;FOLD SLIN P127 Vel=2 m/s CPDAT127 Tool[4]:Microflown3D Base[2]:straight_sol;%{PE}
;FOLD Parameters ;%{h}
;Params IlfProvider=kukaroboter.basistech.inlineforms.movement.spline; Kuka.IsGlobalPoint=False; Kuka.PointName=P127; Kuka.BlendingEnabled=False; Kuka.MoveDataName=CPDAT127; Kuka.VelocityPath=2.000; Kuka.VelocityFieldEnabled=True; Kuka.ColDetectFieldEnabled=True; Kuka.CurrentCDSetIndex=0; Kuka.MovementParameterFieldEnabled=True; IlfCommand=SLIN
;ENDFOLD
SLIN XP127 WITH $VEL = SVEL_CP(2.0, , LCPDAT127),$TOOL = STOOL2(FP127),$BASE = SBASE(FP127.BASE_NO),$IPO_MODE = SIPO_MODE(FP127.IPO_FRAME),$LOAD = SLOAD(FP127.TOOL_NO),$ACC = SACC_CP(LCPDAT127),$ORI_TYPE = SORI_TYP(LCPDAT127),$APO = SAPO(LCPDAT127),$JERK = SJERK(LCPDAT127),$COLLMON_TOL_PRO[1] = USE_CM_PRO_VALUES(0)
;ENDFOLD

;FOLD SLIN P128 Vel=2 m/s CPDAT128 Tool[4]:Microflown3D Base[2]:straight_sol;%{PE}
;FOLD Parameters ;%{h}
;Params IlfProvider=kukaroboter.basistech.inlineforms.movement.spline; Kuka.IsGlobalPoint=False; Kuka.PointName=P128; Kuka.BlendingEnabled=False; Kuka.MoveDataName=CPDAT128; Kuka.VelocityPath=2.000; Kuka.VelocityFieldEnabled=True; Kuka.ColDetectFieldEnabled=True; Kuka.CurrentCDSetIndex=0; Kuka.MovementParameterFieldEnabled=True; IlfCommand=SLIN
;ENDFOLD
SLIN XP128 WITH $VEL = SVEL_CP(2.0, , LCPDAT128),$TOOL = STOOL2(FP128),$BASE = SBASE(FP128.BASE_NO),$IPO_MODE = SIPO_MODE(FP128.IPO_FRAME),$LOAD = SLOAD(FP128.TOOL_NO),$ACC = SACC_CP(LCPDAT128),$ORI_TYPE = SORI_TYP(LCPDAT128),$APO = SAPO(LCPDAT128),$JERK = SJERK(LCPDAT128),$COLLMON_TOL_PRO[1] = USE_CM_PRO_VALUES(0)
;ENDFOLD

;FOLD SLIN P129 Vel=2 m/s CPDAT129 Tool[4]:Microflown3D Base[2]:straight_sol;%{PE}
;FOLD Parameters ;%{h}
;Params IlfProvider=kukaroboter.basistech.inlineforms.movement.spline; Kuka.IsGlobalPoint=False; Kuka.PointName=P129; Kuka.BlendingEnabled=False; Kuka.MoveDataName=CPDAT129; Kuka.VelocityPath=2.000; Kuka.VelocityFieldEnabled=True; Kuka.ColDetectFieldEnabled=True; Kuka.CurrentCDSetIndex=0; Kuka.MovementParameterFieldEnabled=True; IlfCommand=SLIN
;ENDFOLD
SLIN XP129 WITH $VEL = SVEL_CP(2.0, , LCPDAT129),$TOOL = STOOL2(FP129),$BASE = SBASE(FP129.BASE_NO),$IPO_MODE = SIPO_MODE(FP129.IPO_FRAME),$LOAD = SLOAD(FP129.TOOL_NO),$ACC = SACC_CP(LCPDAT129),$ORI_TYPE = SORI_TYP(LCPDAT129),$APO = SAPO(LCPDAT129),$JERK = SJERK(LCPDAT129),$COLLMON_TOL_PRO[1] = USE_CM_PRO_VALUES(0)
;ENDFOLD

;FOLD SLIN P130 Vel=2 m/s CPDAT130 Tool[4]:Microflown3D Base[2]:straight_sol;%{PE}
;FOLD Parameters ;%{h}
;Params IlfProvider=kukaroboter.basistech.inlineforms.movement.spline; Kuka.IsGlobalPoint=False; Kuka.PointName=P130; Kuka.BlendingEnabled=False; Kuka.MoveDataName=CPDAT130; Kuka.VelocityPath=2.000; Kuka.VelocityFieldEnabled=True; Kuka.ColDetectFieldEnabled=True; Kuka.CurrentCDSetIndex=0; Kuka.MovementParameterFieldEnabled=True; IlfCommand=SLIN
;ENDFOLD
SLIN XP130 WITH $VEL = SVEL_CP(2.0, , LCPDAT130),$TOOL = STOOL2(FP130),$BASE = SBASE(FP130.BASE_NO),$IPO_MODE = SIPO_MODE(FP130.IPO_FRAME),$LOAD = SLOAD(FP130.TOOL_NO),$ACC = SACC_CP(LCPDAT130),$ORI_TYPE = SORI_TYP(LCPDAT130),$APO = SAPO(LCPDAT130),$JERK = SJERK(LCPDAT130),$COLLMON_TOL_PRO[1] = USE_CM_PRO_VALUES(0)
;ENDFOLD

;FOLD SLIN P131 Vel=2 m/s CPDAT131 Tool[4]:Microflown3D Base[2]:straight_sol;%{PE}
;FOLD Parameters ;%{h}
;Params IlfProvider=kukaroboter.basistech.inlineforms.movement.spline; Kuka.IsGlobalPoint=False; Kuka.PointName=P131; Kuka.BlendingEnabled=False; Kuka.MoveDataName=CPDAT131; Kuka.VelocityPath=2.000; Kuka.VelocityFieldEnabled=True; Kuka.ColDetectFieldEnabled=True; Kuka.CurrentCDSetIndex=0; Kuka.MovementParameterFieldEnabled=True; IlfCommand=SLIN
;ENDFOLD
SLIN XP131 WITH $VEL = SVEL_CP(2.0, , LCPDAT131),$TOOL = STOOL2(FP131),$BASE = SBASE(FP131.BASE_NO),$IPO_MODE = SIPO_MODE(FP131.IPO_FRAME),$LOAD = SLOAD(FP131.TOOL_NO),$ACC = SACC_CP(LCPDAT131),$ORI_TYPE = SORI_TYP(LCPDAT131),$APO = SAPO(LCPDAT131),$JERK = SJERK(LCPDAT131),$COLLMON_TOL_PRO[1] = USE_CM_PRO_VALUES(0)
;ENDFOLD

;FOLD SLIN P132 Vel=2 m/s CPDAT132 Tool[4]:Microflown3D Base[2]:straight_sol;%{PE}
;FOLD Parameters ;%{h}
;Params IlfProvider=kukaroboter.basistech.inlineforms.movement.spline; Kuka.IsGlobalPoint=False; Kuka.PointName=P132; Kuka.BlendingEnabled=False; Kuka.MoveDataName=CPDAT132; Kuka.VelocityPath=2.000; Kuka.VelocityFieldEnabled=True; Kuka.ColDetectFieldEnabled=True; Kuka.CurrentCDSetIndex=0; Kuka.MovementParameterFieldEnabled=True; IlfCommand=SLIN
;ENDFOLD
SLIN XP132 WITH $VEL = SVEL_CP(2.0, , LCPDAT132),$TOOL = STOOL2(FP132),$BASE = SBASE(FP132.BASE_NO),$IPO_MODE = SIPO_MODE(FP132.IPO_FRAME),$LOAD = SLOAD(FP132.TOOL_NO),$ACC = SACC_CP(LCPDAT132),$ORI_TYPE = SORI_TYP(LCPDAT132),$APO = SAPO(LCPDAT132),$JERK = SJERK(LCPDAT132),$COLLMON_TOL_PRO[1] = USE_CM_PRO_VALUES(0)
;ENDFOLD

;FOLD SLIN P133 Vel=2 m/s CPDAT133 Tool[4]:Microflown3D Base[2]:straight_sol;%{PE}
;FOLD Parameters ;%{h}
;Params IlfProvider=kukaroboter.basistech.inlineforms.movement.spline; Kuka.IsGlobalPoint=False; Kuka.PointName=P133; Kuka.BlendingEnabled=False; Kuka.MoveDataName=CPDAT133; Kuka.VelocityPath=2.000; Kuka.VelocityFieldEnabled=True; Kuka.ColDetectFieldEnabled=True; Kuka.CurrentCDSetIndex=0; Kuka.MovementParameterFieldEnabled=True; IlfCommand=SLIN
;ENDFOLD
SLIN XP133 WITH $VEL = SVEL_CP(2.0, , LCPDAT133),$TOOL = STOOL2(FP133),$BASE = SBASE(FP133.BASE_NO),$IPO_MODE = SIPO_MODE(FP133.IPO_FRAME),$LOAD = SLOAD(FP133.TOOL_NO),$ACC = SACC_CP(LCPDAT133),$ORI_TYPE = SORI_TYP(LCPDAT133),$APO = SAPO(LCPDAT133),$JERK = SJERK(LCPDAT133),$COLLMON_TOL_PRO[1] = USE_CM_PRO_VALUES(0)
;ENDFOLD

;FOLD SLIN P134 Vel=2 m/s CPDAT134 Tool[4]:Microflown3D Base[2]:straight_sol;%{PE}
;FOLD Parameters ;%{h}
;Params IlfProvider=kukaroboter.basistech.inlineforms.movement.spline; Kuka.IsGlobalPoint=False; Kuka.PointName=P134; Kuka.BlendingEnabled=False; Kuka.MoveDataName=CPDAT134; Kuka.VelocityPath=2.000; Kuka.VelocityFieldEnabled=True; Kuka.ColDetectFieldEnabled=True; Kuka.CurrentCDSetIndex=0; Kuka.MovementParameterFieldEnabled=True; IlfCommand=SLIN
;ENDFOLD
SLIN XP134 WITH $VEL = SVEL_CP(2.0, , LCPDAT134),$TOOL = STOOL2(FP134),$BASE = SBASE(FP134.BASE_NO),$IPO_MODE = SIPO_MODE(FP134.IPO_FRAME),$LOAD = SLOAD(FP134.TOOL_NO),$ACC = SACC_CP(LCPDAT134),$ORI_TYPE = SORI_TYP(LCPDAT134),$APO = SAPO(LCPDAT134),$JERK = SJERK(LCPDAT134),$COLLMON_TOL_PRO[1] = USE_CM_PRO_VALUES(0)
;ENDFOLD

;FOLD SLIN P135 Vel=1 m/s CPDAT135 Tool[4]:Microflown3D Base[2]:straight_sol;%{PE}
;FOLD Parameters ;%{h}
;Params IlfProvider=kukaroboter.basistech.inlineforms.movement.spline; Kuka.IsGlobalPoint=False; Kuka.PointName=P135; Kuka.BlendingEnabled=False; Kuka.MoveDataName=CPDAT135; Kuka.VelocityPath=1.000; Kuka.VelocityFieldEnabled=True; Kuka.ColDetectFieldEnabled=True; Kuka.CurrentCDSetIndex=0; Kuka.MovementParameterFieldEnabled=True; IlfCommand=SLIN
;ENDFOLD
SLIN XP135 WITH $VEL = SVEL_CP(2.0, , LCPDAT135),$TOOL = STOOL2(FP135),$BASE = SBASE(FP135.BASE_NO),$IPO_MODE = SIPO_MODE(FP135.IPO_FRAME),$LOAD = SLOAD(FP135.TOOL_NO),$ACC = SACC_CP(LCPDAT135),$ORI_TYPE = SORI_TYP(LCPDAT135),$APO = SAPO(LCPDAT135),$JERK = SJERK(LCPDAT135),$COLLMON_TOL_PRO[1] = USE_CM_PRO_VALUES(0)
;ENDFOLD

;FOLD SLIN P136 Vel=1 m/s CPDAT136 Tool[4]:Microflown3D Base[2]:straight_sol;%{PE}
;FOLD Parameters ;%{h}
;Params IlfProvider=kukaroboter.basistech.inlineforms.movement.spline; Kuka.IsGlobalPoint=False; Kuka.PointName=P136; Kuka.BlendingEnabled=False; Kuka.MoveDataName=CPDAT136; Kuka.VelocityPath=1.000; Kuka.VelocityFieldEnabled=True; Kuka.ColDetectFieldEnabled=True; Kuka.CurrentCDSetIndex=0; Kuka.MovementParameterFieldEnabled=True; IlfCommand=SLIN
;ENDFOLD
SLIN XP136 WITH $VEL = SVEL_CP(2.0, , LCPDAT136),$TOOL = STOOL2(FP136),$BASE = SBASE(FP136.BASE_NO),$IPO_MODE = SIPO_MODE(FP136.IPO_FRAME),$LOAD = SLOAD(FP136.TOOL_NO),$ACC = SACC_CP(LCPDAT136),$ORI_TYPE = SORI_TYP(LCPDAT136),$APO = SAPO(LCPDAT136),$JERK = SJERK(LCPDAT136),$COLLMON_TOL_PRO[1] = USE_CM_PRO_VALUES(0)
;ENDFOLD

;FOLD SLIN P137 Vel=2 m/s CPDAT137 Tool[4]:Microflown3D Base[2]:straight_sol;%{PE}
;FOLD Parameters ;%{h}
;Params IlfProvider=kukaroboter.basistech.inlineforms.movement.spline; Kuka.IsGlobalPoint=False; Kuka.PointName=P137; Kuka.BlendingEnabled=False; Kuka.MoveDataName=CPDAT137; Kuka.VelocityPath=2.000; Kuka.VelocityFieldEnabled=True; Kuka.ColDetectFieldEnabled=True; Kuka.CurrentCDSetIndex=0; Kuka.MovementParameterFieldEnabled=True; IlfCommand=SLIN
;ENDFOLD
SLIN XP137 WITH $VEL = SVEL_CP(2.0, , LCPDAT137),$TOOL = STOOL2(FP137),$BASE = SBASE(FP137.BASE_NO),$IPO_MODE = SIPO_MODE(FP137.IPO_FRAME),$LOAD = SLOAD(FP137.TOOL_NO),$ACC = SACC_CP(LCPDAT137),$ORI_TYPE = SORI_TYP(LCPDAT137),$APO = SAPO(LCPDAT137),$JERK = SJERK(LCPDAT137),$COLLMON_TOL_PRO[1] = USE_CM_PRO_VALUES(0)
;ENDFOLD

;FOLD SLIN P138 Vel=2 m/s CPDAT138 Tool[4]:Microflown3D Base[2]:straight_sol;%{PE}
;FOLD Parameters ;%{h}
;Params IlfProvider=kukaroboter.basistech.inlineforms.movement.spline; Kuka.IsGlobalPoint=False; Kuka.PointName=P138; Kuka.BlendingEnabled=False; Kuka.MoveDataName=CPDAT138; Kuka.VelocityPath=2.000; Kuka.VelocityFieldEnabled=True; Kuka.ColDetectFieldEnabled=True; Kuka.CurrentCDSetIndex=0; Kuka.MovementParameterFieldEnabled=True; IlfCommand=SLIN
;ENDFOLD
SLIN XP138 WITH $VEL = SVEL_CP(2.0, , LCPDAT138),$TOOL = STOOL2(FP138),$BASE = SBASE(FP138.BASE_NO),$IPO_MODE = SIPO_MODE(FP138.IPO_FRAME),$LOAD = SLOAD(FP138.TOOL_NO),$ACC = SACC_CP(LCPDAT138),$ORI_TYPE = SORI_TYP(LCPDAT138),$APO = SAPO(LCPDAT138),$JERK = SJERK(LCPDAT138),$COLLMON_TOL_PRO[1] = USE_CM_PRO_VALUES(0)
;ENDFOLD

;FOLD SLIN P139 Vel=2 m/s CPDAT139 Tool[4]:Microflown3D Base[2]:straight_sol;%{PE}
;FOLD Parameters ;%{h}
;Params IlfProvider=kukaroboter.basistech.inlineforms.movement.spline; Kuka.IsGlobalPoint=False; Kuka.PointName=P139; Kuka.BlendingEnabled=False; Kuka.MoveDataName=CPDAT139; Kuka.VelocityPath=2.000; Kuka.VelocityFieldEnabled=True; Kuka.ColDetectFieldEnabled=True; Kuka.CurrentCDSetIndex=0; Kuka.MovementParameterFieldEnabled=True; IlfCommand=SLIN
;ENDFOLD
SLIN XP139 WITH $VEL = SVEL_CP(2.0, , LCPDAT139),$TOOL = STOOL2(FP139),$BASE = SBASE(FP139.BASE_NO),$IPO_MODE = SIPO_MODE(FP139.IPO_FRAME),$LOAD = SLOAD(FP139.TOOL_NO),$ACC = SACC_CP(LCPDAT139),$ORI_TYPE = SORI_TYP(LCPDAT139),$APO = SAPO(LCPDAT139),$JERK = SJERK(LCPDAT139),$COLLMON_TOL_PRO[1] = USE_CM_PRO_VALUES(0)
;ENDFOLD

;FOLD SLIN P140 Vel=2 m/s CPDAT140 Tool[4]:Microflown3D Base[2]:straight_sol;%{PE}
;FOLD Parameters ;%{h}
;Params IlfProvider=kukaroboter.basistech.inlineforms.movement.spline; Kuka.IsGlobalPoint=False; Kuka.PointName=P140; Kuka.BlendingEnabled=False; Kuka.MoveDataName=CPDAT140; Kuka.VelocityPath=2.000; Kuka.VelocityFieldEnabled=True; Kuka.ColDetectFieldEnabled=True; Kuka.CurrentCDSetIndex=0; Kuka.MovementParameterFieldEnabled=True; IlfCommand=SLIN
;ENDFOLD
SLIN XP140 WITH $VEL = SVEL_CP(2.0, , LCPDAT140),$TOOL = STOOL2(FP140),$BASE = SBASE(FP140.BASE_NO),$IPO_MODE = SIPO_MODE(FP140.IPO_FRAME),$LOAD = SLOAD(FP140.TOOL_NO),$ACC = SACC_CP(LCPDAT140),$ORI_TYPE = SORI_TYP(LCPDAT140),$APO = SAPO(LCPDAT140),$JERK = SJERK(LCPDAT140),$COLLMON_TOL_PRO[1] = USE_CM_PRO_VALUES(0)
;ENDFOLD

;FOLD SLIN P141 Vel=2 m/s CPDAT141 Tool[4]:Microflown3D Base[2]:straight_sol;%{PE}
;FOLD Parameters ;%{h}
;Params IlfProvider=kukaroboter.basistech.inlineforms.movement.spline; Kuka.IsGlobalPoint=False; Kuka.PointName=P141; Kuka.BlendingEnabled=False; Kuka.MoveDataName=CPDAT141; Kuka.VelocityPath=2.000; Kuka.VelocityFieldEnabled=True; Kuka.ColDetectFieldEnabled=True; Kuka.CurrentCDSetIndex=0; Kuka.MovementParameterFieldEnabled=True; IlfCommand=SLIN
;ENDFOLD
SLIN XP141 WITH $VEL = SVEL_CP(2.0, , LCPDAT141),$TOOL = STOOL2(FP141),$BASE = SBASE(FP141.BASE_NO),$IPO_MODE = SIPO_MODE(FP141.IPO_FRAME),$LOAD = SLOAD(FP141.TOOL_NO),$ACC = SACC_CP(LCPDAT141),$ORI_TYPE = SORI_TYP(LCPDAT141),$APO = SAPO(LCPDAT141),$JERK = SJERK(LCPDAT141),$COLLMON_TOL_PRO[1] = USE_CM_PRO_VALUES(0)
;ENDFOLD

;FOLD SLIN P142 Vel=2 m/s CPDAT142 Tool[4]:Microflown3D Base[2]:straight_sol;%{PE}
;FOLD Parameters ;%{h}
;Params IlfProvider=kukaroboter.basistech.inlineforms.movement.spline; Kuka.IsGlobalPoint=False; Kuka.PointName=P142; Kuka.BlendingEnabled=False; Kuka.MoveDataName=CPDAT142; Kuka.VelocityPath=2.000; Kuka.VelocityFieldEnabled=True; Kuka.ColDetectFieldEnabled=True; Kuka.CurrentCDSetIndex=0; Kuka.MovementParameterFieldEnabled=True; IlfCommand=SLIN
;ENDFOLD
SLIN XP142 WITH $VEL = SVEL_CP(2.0, , LCPDAT142),$TOOL = STOOL2(FP142),$BASE = SBASE(FP142.BASE_NO),$IPO_MODE = SIPO_MODE(FP142.IPO_FRAME),$LOAD = SLOAD(FP142.TOOL_NO),$ACC = SACC_CP(LCPDAT142),$ORI_TYPE = SORI_TYP(LCPDAT142),$APO = SAPO(LCPDAT142),$JERK = SJERK(LCPDAT142),$COLLMON_TOL_PRO[1] = USE_CM_PRO_VALUES(0)
;ENDFOLD

;FOLD SLIN P143 Vel=2 m/s CPDAT143 Tool[4]:Microflown3D Base[2]:straight_sol;%{PE}
;FOLD Parameters ;%{h}
;Params IlfProvider=kukaroboter.basistech.inlineforms.movement.spline; Kuka.IsGlobalPoint=False; Kuka.PointName=P143; Kuka.BlendingEnabled=False; Kuka.MoveDataName=CPDAT143; Kuka.VelocityPath=2.000; Kuka.VelocityFieldEnabled=True; Kuka.ColDetectFieldEnabled=True; Kuka.CurrentCDSetIndex=0; Kuka.MovementParameterFieldEnabled=True; IlfCommand=SLIN
;ENDFOLD
SLIN XP143 WITH $VEL = SVEL_CP(2.0, , LCPDAT143),$TOOL = STOOL2(FP143),$BASE = SBASE(FP143.BASE_NO),$IPO_MODE = SIPO_MODE(FP143.IPO_FRAME),$LOAD = SLOAD(FP143.TOOL_NO),$ACC = SACC_CP(LCPDAT143),$ORI_TYPE = SORI_TYP(LCPDAT143),$APO = SAPO(LCPDAT143),$JERK = SJERK(LCPDAT143),$COLLMON_TOL_PRO[1] = USE_CM_PRO_VALUES(0)
;ENDFOLD

;FOLD SLIN P144 Vel=2 m/s CPDAT144 Tool[4]:Microflown3D Base[2]:straight_sol;%{PE}
;FOLD Parameters ;%{h}
;Params IlfProvider=kukaroboter.basistech.inlineforms.movement.spline; Kuka.IsGlobalPoint=False; Kuka.PointName=P144; Kuka.BlendingEnabled=False; Kuka.MoveDataName=CPDAT144; Kuka.VelocityPath=2.000; Kuka.VelocityFieldEnabled=True; Kuka.ColDetectFieldEnabled=True; Kuka.CurrentCDSetIndex=0; Kuka.MovementParameterFieldEnabled=True; IlfCommand=SLIN
;ENDFOLD
SLIN XP144 WITH $VEL = SVEL_CP(2.0, , LCPDAT144),$TOOL = STOOL2(FP144),$BASE = SBASE(FP144.BASE_NO),$IPO_MODE = SIPO_MODE(FP144.IPO_FRAME),$LOAD = SLOAD(FP144.TOOL_NO),$ACC = SACC_CP(LCPDAT144),$ORI_TYPE = SORI_TYP(LCPDAT144),$APO = SAPO(LCPDAT144),$JERK = SJERK(LCPDAT144),$COLLMON_TOL_PRO[1] = USE_CM_PRO_VALUES(0)
;ENDFOLD

;FOLD SLIN P145 Vel=2 m/s CPDAT145 Tool[4]:Microflown3D Base[2]:straight_sol;%{PE}
;FOLD Parameters ;%{h}
;Params IlfProvider=kukaroboter.basistech.inlineforms.movement.spline; Kuka.IsGlobalPoint=False; Kuka.PointName=P145; Kuka.BlendingEnabled=False; Kuka.MoveDataName=CPDAT145; Kuka.VelocityPath=2.000; Kuka.VelocityFieldEnabled=True; Kuka.ColDetectFieldEnabled=True; Kuka.CurrentCDSetIndex=0; Kuka.MovementParameterFieldEnabled=True; IlfCommand=SLIN
;ENDFOLD
SLIN XP145 WITH $VEL = SVEL_CP(2.0, , LCPDAT145),$TOOL = STOOL2(FP145),$BASE = SBASE(FP145.BASE_NO),$IPO_MODE = SIPO_MODE(FP145.IPO_FRAME),$LOAD = SLOAD(FP145.TOOL_NO),$ACC = SACC_CP(LCPDAT145),$ORI_TYPE = SORI_TYP(LCPDAT145),$APO = SAPO(LCPDAT145),$JERK = SJERK(LCPDAT145),$COLLMON_TOL_PRO[1] = USE_CM_PRO_VALUES(0)
;ENDFOLD

;FOLD SLIN P146 Vel=2 m/s CPDAT146 Tool[4]:Microflown3D Base[2]:straight_sol;%{PE}
;FOLD Parameters ;%{h}
;Params IlfProvider=kukaroboter.basistech.inlineforms.movement.spline; Kuka.IsGlobalPoint=False; Kuka.PointName=P146; Kuka.BlendingEnabled=False; Kuka.MoveDataName=CPDAT146; Kuka.VelocityPath=2.000; Kuka.VelocityFieldEnabled=True; Kuka.ColDetectFieldEnabled=True; Kuka.CurrentCDSetIndex=0; Kuka.MovementParameterFieldEnabled=True; IlfCommand=SLIN
;ENDFOLD
SLIN XP146 WITH $VEL = SVEL_CP(2.0, , LCPDAT146),$TOOL = STOOL2(FP146),$BASE = SBASE(FP146.BASE_NO),$IPO_MODE = SIPO_MODE(FP146.IPO_FRAME),$LOAD = SLOAD(FP146.TOOL_NO),$ACC = SACC_CP(LCPDAT146),$ORI_TYPE = SORI_TYP(LCPDAT146),$APO = SAPO(LCPDAT146),$JERK = SJERK(LCPDAT146),$COLLMON_TOL_PRO[1] = USE_CM_PRO_VALUES(0)
;ENDFOLD

;FOLD SLIN P147 Vel=2 m/s CPDAT147 Tool[4]:Microflown3D Base[2]:straight_sol;%{PE}
;FOLD Parameters ;%{h}
;Params IlfProvider=kukaroboter.basistech.inlineforms.movement.spline; Kuka.IsGlobalPoint=False; Kuka.PointName=P147; Kuka.BlendingEnabled=False; Kuka.MoveDataName=CPDAT147; Kuka.VelocityPath=2.000; Kuka.VelocityFieldEnabled=True; Kuka.ColDetectFieldEnabled=True; Kuka.CurrentCDSetIndex=0; Kuka.MovementParameterFieldEnabled=True; IlfCommand=SLIN
;ENDFOLD
SLIN XP147 WITH $VEL = SVEL_CP(2.0, , LCPDAT147),$TOOL = STOOL2(FP147),$BASE = SBASE(FP147.BASE_NO),$IPO_MODE = SIPO_MODE(FP147.IPO_FRAME),$LOAD = SLOAD(FP147.TOOL_NO),$ACC = SACC_CP(LCPDAT147),$ORI_TYPE = SORI_TYP(LCPDAT147),$APO = SAPO(LCPDAT147),$JERK = SJERK(LCPDAT147),$COLLMON_TOL_PRO[1] = USE_CM_PRO_VALUES(0)
;ENDFOLD

;FOLD SLIN P148 Vel=2 m/s CPDAT148 Tool[4]:Microflown3D Base[2]:straight_sol;%{PE}
;FOLD Parameters ;%{h}
;Params IlfProvider=kukaroboter.basistech.inlineforms.movement.spline; Kuka.IsGlobalPoint=False; Kuka.PointName=P148; Kuka.BlendingEnabled=False; Kuka.MoveDataName=CPDAT148; Kuka.VelocityPath=2.000; Kuka.VelocityFieldEnabled=True; Kuka.ColDetectFieldEnabled=True; Kuka.CurrentCDSetIndex=0; Kuka.MovementParameterFieldEnabled=True; IlfCommand=SLIN
;ENDFOLD
SLIN XP148 WITH $VEL = SVEL_CP(2.0, , LCPDAT148),$TOOL = STOOL2(FP148),$BASE = SBASE(FP148.BASE_NO),$IPO_MODE = SIPO_MODE(FP148.IPO_FRAME),$LOAD = SLOAD(FP148.TOOL_NO),$ACC = SACC_CP(LCPDAT148),$ORI_TYPE = SORI_TYP(LCPDAT148),$APO = SAPO(LCPDAT148),$JERK = SJERK(LCPDAT148),$COLLMON_TOL_PRO[1] = USE_CM_PRO_VALUES(0)
;ENDFOLD

;FOLD SLIN P149 Vel=2 m/s CPDAT149 Tool[4]:Microflown3D Base[2]:straight_sol;%{PE}
;FOLD Parameters ;%{h}
;Params IlfProvider=kukaroboter.basistech.inlineforms.movement.spline; Kuka.IsGlobalPoint=False; Kuka.PointName=P149; Kuka.BlendingEnabled=False; Kuka.MoveDataName=CPDAT149; Kuka.VelocityPath=2.000; Kuka.VelocityFieldEnabled=True; Kuka.ColDetectFieldEnabled=True; Kuka.CurrentCDSetIndex=0; Kuka.MovementParameterFieldEnabled=True; IlfCommand=SLIN
;ENDFOLD
SLIN XP149 WITH $VEL = SVEL_CP(2.0, , LCPDAT149),$TOOL = STOOL2(FP149),$BASE = SBASE(FP149.BASE_NO),$IPO_MODE = SIPO_MODE(FP149.IPO_FRAME),$LOAD = SLOAD(FP149.TOOL_NO),$ACC = SACC_CP(LCPDAT149),$ORI_TYPE = SORI_TYP(LCPDAT149),$APO = SAPO(LCPDAT149),$JERK = SJERK(LCPDAT149),$COLLMON_TOL_PRO[1] = USE_CM_PRO_VALUES(0)
;ENDFOLD

;FOLD SLIN P150 Vel=2 m/s CPDAT150 Tool[4]:Microflown3D Base[2]:straight_sol;%{PE}
;FOLD Parameters ;%{h}
;Params IlfProvider=kukaroboter.basistech.inlineforms.movement.spline; Kuka.IsGlobalPoint=False; Kuka.PointName=P150; Kuka.BlendingEnabled=False; Kuka.MoveDataName=CPDAT150; Kuka.VelocityPath=2.000; Kuka.VelocityFieldEnabled=True; Kuka.ColDetectFieldEnabled=True; Kuka.CurrentCDSetIndex=0; Kuka.MovementParameterFieldEnabled=True; IlfCommand=SLIN
;ENDFOLD
SLIN XP150 WITH $VEL = SVEL_CP(2.0, , LCPDAT150),$TOOL = STOOL2(FP150),$BASE = SBASE(FP150.BASE_NO),$IPO_MODE = SIPO_MODE(FP150.IPO_FRAME),$LOAD = SLOAD(FP150.TOOL_NO),$ACC = SACC_CP(LCPDAT150),$ORI_TYPE = SORI_TYP(LCPDAT150),$APO = SAPO(LCPDAT150),$JERK = SJERK(LCPDAT150),$COLLMON_TOL_PRO[1] = USE_CM_PRO_VALUES(0)
;ENDFOLD

;FOLD SLIN P151 Vel=2 m/s CPDAT151 Tool[4]:Microflown3D Base[2]:straight_sol;%{PE}
;FOLD Parameters ;%{h}
;Params IlfProvider=kukaroboter.basistech.inlineforms.movement.spline; Kuka.IsGlobalPoint=False; Kuka.PointName=P151; Kuka.BlendingEnabled=False; Kuka.MoveDataName=CPDAT151; Kuka.VelocityPath=2.000; Kuka.VelocityFieldEnabled=True; Kuka.ColDetectFieldEnabled=True; Kuka.CurrentCDSetIndex=0; Kuka.MovementParameterFieldEnabled=True; IlfCommand=SLIN
;ENDFOLD
SLIN XP151 WITH $VEL = SVEL_CP(2.0, , LCPDAT151),$TOOL = STOOL2(FP151),$BASE = SBASE(FP151.BASE_NO),$IPO_MODE = SIPO_MODE(FP151.IPO_FRAME),$LOAD = SLOAD(FP151.TOOL_NO),$ACC = SACC_CP(LCPDAT151),$ORI_TYPE = SORI_TYP(LCPDAT151),$APO = SAPO(LCPDAT151),$JERK = SJERK(LCPDAT151),$COLLMON_TOL_PRO[1] = USE_CM_PRO_VALUES(0)
;ENDFOLD

;FOLD SLIN P152 Vel=2 m/s CPDAT152 Tool[4]:Microflown3D Base[2]:straight_sol;%{PE}
;FOLD Parameters ;%{h}
;Params IlfProvider=kukaroboter.basistech.inlineforms.movement.spline; Kuka.IsGlobalPoint=False; Kuka.PointName=P152; Kuka.BlendingEnabled=False; Kuka.MoveDataName=CPDAT152; Kuka.VelocityPath=2.000; Kuka.VelocityFieldEnabled=True; Kuka.ColDetectFieldEnabled=True; Kuka.CurrentCDSetIndex=0; Kuka.MovementParameterFieldEnabled=True; IlfCommand=SLIN
;ENDFOLD
SLIN XP152 WITH $VEL = SVEL_CP(2.0, , LCPDAT152),$TOOL = STOOL2(FP152),$BASE = SBASE(FP152.BASE_NO),$IPO_MODE = SIPO_MODE(FP152.IPO_FRAME),$LOAD = SLOAD(FP152.TOOL_NO),$ACC = SACC_CP(LCPDAT152),$ORI_TYPE = SORI_TYP(LCPDAT152),$APO = SAPO(LCPDAT152),$JERK = SJERK(LCPDAT152),$COLLMON_TOL_PRO[1] = USE_CM_PRO_VALUES(0)
;ENDFOLD

;FOLD SLIN P153 Vel=2 m/s CPDAT153 Tool[4]:Microflown3D Base[2]:straight_sol;%{PE}
;FOLD Parameters ;%{h}
;Params IlfProvider=kukaroboter.basistech.inlineforms.movement.spline; Kuka.IsGlobalPoint=False; Kuka.PointName=P153; Kuka.BlendingEnabled=False; Kuka.MoveDataName=CPDAT153; Kuka.VelocityPath=2.000; Kuka.VelocityFieldEnabled=True; Kuka.ColDetectFieldEnabled=True; Kuka.CurrentCDSetIndex=0; Kuka.MovementParameterFieldEnabled=True; IlfCommand=SLIN
;ENDFOLD
SLIN XP153 WITH $VEL = SVEL_CP(2.0, , LCPDAT153),$TOOL = STOOL2(FP153),$BASE = SBASE(FP153.BASE_NO),$IPO_MODE = SIPO_MODE(FP153.IPO_FRAME),$LOAD = SLOAD(FP153.TOOL_NO),$ACC = SACC_CP(LCPDAT153),$ORI_TYPE = SORI_TYP(LCPDAT153),$APO = SAPO(LCPDAT153),$JERK = SJERK(LCPDAT153),$COLLMON_TOL_PRO[1] = USE_CM_PRO_VALUES(0)
;ENDFOLD

;FOLD SLIN P154 Vel=2 m/s CPDAT154 Tool[4]:Microflown3D Base[2]:straight_sol;%{PE}
;FOLD Parameters ;%{h}
;Params IlfProvider=kukaroboter.basistech.inlineforms.movement.spline; Kuka.IsGlobalPoint=False; Kuka.PointName=P154; Kuka.BlendingEnabled=False; Kuka.MoveDataName=CPDAT154; Kuka.VelocityPath=2.000; Kuka.VelocityFieldEnabled=True; Kuka.ColDetectFieldEnabled=True; Kuka.CurrentCDSetIndex=0; Kuka.MovementParameterFieldEnabled=True; IlfCommand=SLIN
;ENDFOLD
SLIN XP154 WITH $VEL = SVEL_CP(2.0, , LCPDAT154),$TOOL = STOOL2(FP154),$BASE = SBASE(FP154.BASE_NO),$IPO_MODE = SIPO_MODE(FP154.IPO_FRAME),$LOAD = SLOAD(FP154.TOOL_NO),$ACC = SACC_CP(LCPDAT154),$ORI_TYPE = SORI_TYP(LCPDAT154),$APO = SAPO(LCPDAT154),$JERK = SJERK(LCPDAT154),$COLLMON_TOL_PRO[1] = USE_CM_PRO_VALUES(0)
;ENDFOLD

;FOLD SLIN P155 Vel=2 m/s CPDAT155 Tool[4]:Microflown3D Base[2]:straight_sol;%{PE}
;FOLD Parameters ;%{h}
;Params IlfProvider=kukaroboter.basistech.inlineforms.movement.spline; Kuka.IsGlobalPoint=False; Kuka.PointName=P155; Kuka.BlendingEnabled=False; Kuka.MoveDataName=CPDAT155; Kuka.VelocityPath=2.000; Kuka.VelocityFieldEnabled=True; Kuka.ColDetectFieldEnabled=True; Kuka.CurrentCDSetIndex=0; Kuka.MovementParameterFieldEnabled=True; IlfCommand=SLIN
;ENDFOLD
SLIN XP155 WITH $VEL = SVEL_CP(2.0, , LCPDAT155),$TOOL = STOOL2(FP155),$BASE = SBASE(FP155.BASE_NO),$IPO_MODE = SIPO_MODE(FP155.IPO_FRAME),$LOAD = SLOAD(FP155.TOOL_NO),$ACC = SACC_CP(LCPDAT155),$ORI_TYPE = SORI_TYP(LCPDAT155),$APO = SAPO(LCPDAT155),$JERK = SJERK(LCPDAT155),$COLLMON_TOL_PRO[1] = USE_CM_PRO_VALUES(0)
;ENDFOLD

;FOLD SLIN P156 Vel=2 m/s CPDAT156 Tool[4]:Microflown3D Base[2]:straight_sol;%{PE}
;FOLD Parameters ;%{h}
;Params IlfProvider=kukaroboter.basistech.inlineforms.movement.spline; Kuka.IsGlobalPoint=False; Kuka.PointName=P156; Kuka.BlendingEnabled=False; Kuka.MoveDataName=CPDAT156; Kuka.VelocityPath=2.000; Kuka.VelocityFieldEnabled=True; Kuka.ColDetectFieldEnabled=True; Kuka.CurrentCDSetIndex=0; Kuka.MovementParameterFieldEnabled=True; IlfCommand=SLIN
;ENDFOLD
SLIN XP156 WITH $VEL = SVEL_CP(2.0, , LCPDAT156),$TOOL = STOOL2(FP156),$BASE = SBASE(FP156.BASE_NO),$IPO_MODE = SIPO_MODE(FP156.IPO_FRAME),$LOAD = SLOAD(FP156.TOOL_NO),$ACC = SACC_CP(LCPDAT156),$ORI_TYPE = SORI_TYP(LCPDAT156),$APO = SAPO(LCPDAT156),$JERK = SJERK(LCPDAT156),$COLLMON_TOL_PRO[1] = USE_CM_PRO_VALUES(0)
;ENDFOLD

;FOLD SLIN P157 Vel=2 m/s CPDAT157 Tool[4]:Microflown3D Base[2]:straight_sol;%{PE}
;FOLD Parameters ;%{h}
;Params IlfProvider=kukaroboter.basistech.inlineforms.movement.spline; Kuka.IsGlobalPoint=False; Kuka.PointName=P157; Kuka.BlendingEnabled=False; Kuka.MoveDataName=CPDAT157; Kuka.VelocityPath=2.000; Kuka.VelocityFieldEnabled=True; Kuka.ColDetectFieldEnabled=True; Kuka.CurrentCDSetIndex=0; Kuka.MovementParameterFieldEnabled=True; IlfCommand=SLIN
;ENDFOLD
SLIN XP157 WITH $VEL = SVEL_CP(2.0, , LCPDAT157),$TOOL = STOOL2(FP157),$BASE = SBASE(FP157.BASE_NO),$IPO_MODE = SIPO_MODE(FP157.IPO_FRAME),$LOAD = SLOAD(FP157.TOOL_NO),$ACC = SACC_CP(LCPDAT157),$ORI_TYPE = SORI_TYP(LCPDAT157),$APO = SAPO(LCPDAT157),$JERK = SJERK(LCPDAT157),$COLLMON_TOL_PRO[1] = USE_CM_PRO_VALUES(0)
;ENDFOLD

;FOLD SLIN P158 Vel=2 m/s CPDAT158 Tool[4]:Microflown3D Base[2]:straight_sol;%{PE}
;FOLD Parameters ;%{h}
;Params IlfProvider=kukaroboter.basistech.inlineforms.movement.spline; Kuka.IsGlobalPoint=False; Kuka.PointName=P158; Kuka.BlendingEnabled=False; Kuka.MoveDataName=CPDAT158; Kuka.VelocityPath=2.000; Kuka.VelocityFieldEnabled=True; Kuka.ColDetectFieldEnabled=True; Kuka.CurrentCDSetIndex=0; Kuka.MovementParameterFieldEnabled=True; IlfCommand=SLIN
;ENDFOLD
SLIN XP158 WITH $VEL = SVEL_CP(2.0, , LCPDAT158),$TOOL = STOOL2(FP158),$BASE = SBASE(FP158.BASE_NO),$IPO_MODE = SIPO_MODE(FP158.IPO_FRAME),$LOAD = SLOAD(FP158.TOOL_NO),$ACC = SACC_CP(LCPDAT158),$ORI_TYPE = SORI_TYP(LCPDAT158),$APO = SAPO(LCPDAT158),$JERK = SJERK(LCPDAT158),$COLLMON_TOL_PRO[1] = USE_CM_PRO_VALUES(0)
;ENDFOLD

;FOLD SLIN P159 Vel=2 m/s CPDAT159 Tool[4]:Microflown3D Base[2]:straight_sol;%{PE}
;FOLD Parameters ;%{h}
;Params IlfProvider=kukaroboter.basistech.inlineforms.movement.spline; Kuka.IsGlobalPoint=False; Kuka.PointName=P159; Kuka.BlendingEnabled=False; Kuka.MoveDataName=CPDAT159; Kuka.VelocityPath=2.000; Kuka.VelocityFieldEnabled=True; Kuka.ColDetectFieldEnabled=True; Kuka.CurrentCDSetIndex=0; Kuka.MovementParameterFieldEnabled=True; IlfCommand=SLIN
;ENDFOLD
SLIN XP159 WITH $VEL = SVEL_CP(2.0, , LCPDAT159),$TOOL = STOOL2(FP159),$BASE = SBASE(FP159.BASE_NO),$IPO_MODE = SIPO_MODE(FP159.IPO_FRAME),$LOAD = SLOAD(FP159.TOOL_NO),$ACC = SACC_CP(LCPDAT159),$ORI_TYPE = SORI_TYP(LCPDAT159),$APO = SAPO(LCPDAT159),$JERK = SJERK(LCPDAT159),$COLLMON_TOL_PRO[1] = USE_CM_PRO_VALUES(0)
;ENDFOLD

;FOLD SLIN P160 Vel=2 m/s CPDAT160 Tool[4]:Microflown3D Base[2]:straight_sol;%{PE}
;FOLD Parameters ;%{h}
;Params IlfProvider=kukaroboter.basistech.inlineforms.movement.spline; Kuka.IsGlobalPoint=False; Kuka.PointName=P160; Kuka.BlendingEnabled=False; Kuka.MoveDataName=CPDAT160; Kuka.VelocityPath=2.000; Kuka.VelocityFieldEnabled=True; Kuka.ColDetectFieldEnabled=True; Kuka.CurrentCDSetIndex=0; Kuka.MovementParameterFieldEnabled=True; IlfCommand=SLIN
;ENDFOLD
SLIN XP160 WITH $VEL = SVEL_CP(2.0, , LCPDAT160),$TOOL = STOOL2(FP160),$BASE = SBASE(FP160.BASE_NO),$IPO_MODE = SIPO_MODE(FP160.IPO_FRAME),$LOAD = SLOAD(FP160.TOOL_NO),$ACC = SACC_CP(LCPDAT160),$ORI_TYPE = SORI_TYP(LCPDAT160),$APO = SAPO(LCPDAT160),$JERK = SJERK(LCPDAT160),$COLLMON_TOL_PRO[1] = USE_CM_PRO_VALUES(0)
;ENDFOLD

;FOLD SLIN P161 Vel=2 m/s CPDAT161 Tool[4]:Microflown3D Base[2]:straight_sol;%{PE}
;FOLD Parameters ;%{h}
;Params IlfProvider=kukaroboter.basistech.inlineforms.movement.spline; Kuka.IsGlobalPoint=False; Kuka.PointName=P161; Kuka.BlendingEnabled=False; Kuka.MoveDataName=CPDAT161; Kuka.VelocityPath=2.000; Kuka.VelocityFieldEnabled=True; Kuka.ColDetectFieldEnabled=True; Kuka.CurrentCDSetIndex=0; Kuka.MovementParameterFieldEnabled=True; IlfCommand=SLIN
;ENDFOLD
SLIN XP161 WITH $VEL = SVEL_CP(2.0, , LCPDAT161),$TOOL = STOOL2(FP161),$BASE = SBASE(FP161.BASE_NO),$IPO_MODE = SIPO_MODE(FP161.IPO_FRAME),$LOAD = SLOAD(FP161.TOOL_NO),$ACC = SACC_CP(LCPDAT161),$ORI_TYPE = SORI_TYP(LCPDAT161),$APO = SAPO(LCPDAT161),$JERK = SJERK(LCPDAT161),$COLLMON_TOL_PRO[1] = USE_CM_PRO_VALUES(0)
;ENDFOLD

;FOLD SLIN P162 Vel=2 m/s CPDAT162 Tool[4]:Microflown3D Base[2]:straight_sol;%{PE}
;FOLD Parameters ;%{h}
;Params IlfProvider=kukaroboter.basistech.inlineforms.movement.spline; Kuka.IsGlobalPoint=False; Kuka.PointName=P162; Kuka.BlendingEnabled=False; Kuka.MoveDataName=CPDAT162; Kuka.VelocityPath=2.000; Kuka.VelocityFieldEnabled=True; Kuka.ColDetectFieldEnabled=True; Kuka.CurrentCDSetIndex=0; Kuka.MovementParameterFieldEnabled=True; IlfCommand=SLIN
;ENDFOLD
SLIN XP162 WITH $VEL = SVEL_CP(2.0, , LCPDAT162),$TOOL = STOOL2(FP162),$BASE = SBASE(FP162.BASE_NO),$IPO_MODE = SIPO_MODE(FP162.IPO_FRAME),$LOAD = SLOAD(FP162.TOOL_NO),$ACC = SACC_CP(LCPDAT162),$ORI_TYPE = SORI_TYP(LCPDAT162),$APO = SAPO(LCPDAT162),$JERK = SJERK(LCPDAT162),$COLLMON_TOL_PRO[1] = USE_CM_PRO_VALUES(0)
;ENDFOLD

;FOLD SLIN P163 Vel=2 m/s CPDAT163 Tool[4]:Microflown3D Base[2]:straight_sol;%{PE}
;FOLD Parameters ;%{h}
;Params IlfProvider=kukaroboter.basistech.inlineforms.movement.spline; Kuka.IsGlobalPoint=False; Kuka.PointName=P163; Kuka.BlendingEnabled=False; Kuka.MoveDataName=CPDAT163; Kuka.VelocityPath=2.000; Kuka.VelocityFieldEnabled=True; Kuka.ColDetectFieldEnabled=True; Kuka.CurrentCDSetIndex=0; Kuka.MovementParameterFieldEnabled=True; IlfCommand=SLIN
;ENDFOLD
SLIN XP163 WITH $VEL = SVEL_CP(2.0, , LCPDAT163),$TOOL = STOOL2(FP163),$BASE = SBASE(FP163.BASE_NO),$IPO_MODE = SIPO_MODE(FP163.IPO_FRAME),$LOAD = SLOAD(FP163.TOOL_NO),$ACC = SACC_CP(LCPDAT163),$ORI_TYPE = SORI_TYP(LCPDAT163),$APO = SAPO(LCPDAT163),$JERK = SJERK(LCPDAT163),$COLLMON_TOL_PRO[1] = USE_CM_PRO_VALUES(0)
;ENDFOLD

;FOLD SLIN P164 Vel=2 m/s CPDAT164 Tool[4]:Microflown3D Base[2]:straight_sol;%{PE}
;FOLD Parameters ;%{h}
;Params IlfProvider=kukaroboter.basistech.inlineforms.movement.spline; Kuka.IsGlobalPoint=False; Kuka.PointName=P164; Kuka.BlendingEnabled=False; Kuka.MoveDataName=CPDAT164; Kuka.VelocityPath=2.000; Kuka.VelocityFieldEnabled=True; Kuka.ColDetectFieldEnabled=True; Kuka.CurrentCDSetIndex=0; Kuka.MovementParameterFieldEnabled=True; IlfCommand=SLIN
;ENDFOLD
SLIN XP164 WITH $VEL = SVEL_CP(2.0, , LCPDAT164),$TOOL = STOOL2(FP164),$BASE = SBASE(FP164.BASE_NO),$IPO_MODE = SIPO_MODE(FP164.IPO_FRAME),$LOAD = SLOAD(FP164.TOOL_NO),$ACC = SACC_CP(LCPDAT164),$ORI_TYPE = SORI_TYP(LCPDAT164),$APO = SAPO(LCPDAT164),$JERK = SJERK(LCPDAT164),$COLLMON_TOL_PRO[1] = USE_CM_PRO_VALUES(0)
;ENDFOLD

;FOLD SLIN P165 Vel=2 m/s CPDAT165 Tool[4]:Microflown3D Base[2]:straight_sol;%{PE}
;FOLD Parameters ;%{h}
;Params IlfProvider=kukaroboter.basistech.inlineforms.movement.spline; Kuka.IsGlobalPoint=False; Kuka.PointName=P165; Kuka.BlendingEnabled=False; Kuka.MoveDataName=CPDAT165; Kuka.VelocityPath=2.000; Kuka.VelocityFieldEnabled=True; Kuka.ColDetectFieldEnabled=True; Kuka.CurrentCDSetIndex=0; Kuka.MovementParameterFieldEnabled=True; IlfCommand=SLIN
;ENDFOLD
SLIN XP165 WITH $VEL = SVEL_CP(2.0, , LCPDAT165),$TOOL = STOOL2(FP165),$BASE = SBASE(FP165.BASE_NO),$IPO_MODE = SIPO_MODE(FP165.IPO_FRAME),$LOAD = SLOAD(FP165.TOOL_NO),$ACC = SACC_CP(LCPDAT165),$ORI_TYPE = SORI_TYP(LCPDAT165),$APO = SAPO(LCPDAT165),$JERK = SJERK(LCPDAT165),$COLLMON_TOL_PRO[1] = USE_CM_PRO_VALUES(0)
;ENDFOLD

;FOLD SLIN P166 Vel=2 m/s CPDAT166 Tool[4]:Microflown3D Base[2]:straight_sol;%{PE}
;FOLD Parameters ;%{h}
;Params IlfProvider=kukaroboter.basistech.inlineforms.movement.spline; Kuka.IsGlobalPoint=False; Kuka.PointName=P166; Kuka.BlendingEnabled=False; Kuka.MoveDataName=CPDAT166; Kuka.VelocityPath=2.000; Kuka.VelocityFieldEnabled=True; Kuka.ColDetectFieldEnabled=True; Kuka.CurrentCDSetIndex=0; Kuka.MovementParameterFieldEnabled=True; IlfCommand=SLIN
;ENDFOLD
SLIN XP166 WITH $VEL = SVEL_CP(2.0, , LCPDAT166),$TOOL = STOOL2(FP166),$BASE = SBASE(FP166.BASE_NO),$IPO_MODE = SIPO_MODE(FP166.IPO_FRAME),$LOAD = SLOAD(FP166.TOOL_NO),$ACC = SACC_CP(LCPDAT166),$ORI_TYPE = SORI_TYP(LCPDAT166),$APO = SAPO(LCPDAT166),$JERK = SJERK(LCPDAT166),$COLLMON_TOL_PRO[1] = USE_CM_PRO_VALUES(0)
;ENDFOLD

;FOLD SLIN P167 Vel=2 m/s CPDAT167 Tool[4]:Microflown3D Base[2]:straight_sol;%{PE}
;FOLD Parameters ;%{h}
;Params IlfProvider=kukaroboter.basistech.inlineforms.movement.spline; Kuka.IsGlobalPoint=False; Kuka.PointName=P167; Kuka.BlendingEnabled=False; Kuka.MoveDataName=CPDAT167; Kuka.VelocityPath=2.000; Kuka.VelocityFieldEnabled=True; Kuka.ColDetectFieldEnabled=True; Kuka.CurrentCDSetIndex=0; Kuka.MovementParameterFieldEnabled=True; IlfCommand=SLIN
;ENDFOLD
SLIN XP167 WITH $VEL = SVEL_CP(2.0, , LCPDAT167),$TOOL = STOOL2(FP167),$BASE = SBASE(FP167.BASE_NO),$IPO_MODE = SIPO_MODE(FP167.IPO_FRAME),$LOAD = SLOAD(FP167.TOOL_NO),$ACC = SACC_CP(LCPDAT167),$ORI_TYPE = SORI_TYP(LCPDAT167),$APO = SAPO(LCPDAT167),$JERK = SJERK(LCPDAT167),$COLLMON_TOL_PRO[1] = USE_CM_PRO_VALUES(0)
;ENDFOLD

;FOLD SLIN P168 Vel=2 m/s CPDAT168 Tool[4]:Microflown3D Base[2]:straight_sol;%{PE}
;FOLD Parameters ;%{h}
;Params IlfProvider=kukaroboter.basistech.inlineforms.movement.spline; Kuka.IsGlobalPoint=False; Kuka.PointName=P168; Kuka.BlendingEnabled=False; Kuka.MoveDataName=CPDAT168; Kuka.VelocityPath=2.000; Kuka.VelocityFieldEnabled=True; Kuka.ColDetectFieldEnabled=True; Kuka.CurrentCDSetIndex=0; Kuka.MovementParameterFieldEnabled=True; IlfCommand=SLIN
;ENDFOLD
SLIN XP168 WITH $VEL = SVEL_CP(2.0, , LCPDAT168),$TOOL = STOOL2(FP168),$BASE = SBASE(FP168.BASE_NO),$IPO_MODE = SIPO_MODE(FP168.IPO_FRAME),$LOAD = SLOAD(FP168.TOOL_NO),$ACC = SACC_CP(LCPDAT168),$ORI_TYPE = SORI_TYP(LCPDAT168),$APO = SAPO(LCPDAT168),$JERK = SJERK(LCPDAT168),$COLLMON_TOL_PRO[1] = USE_CM_PRO_VALUES(0)
;ENDFOLD

;FOLD SLIN P169 Vel=2 m/s CPDAT169 Tool[4]:Microflown3D Base[2]:straight_sol;%{PE}
;FOLD Parameters ;%{h}
;Params IlfProvider=kukaroboter.basistech.inlineforms.movement.spline; Kuka.IsGlobalPoint=False; Kuka.PointName=P169; Kuka.BlendingEnabled=False; Kuka.MoveDataName=CPDAT169; Kuka.VelocityPath=2.000; Kuka.VelocityFieldEnabled=True; Kuka.ColDetectFieldEnabled=True; Kuka.CurrentCDSetIndex=0; Kuka.MovementParameterFieldEnabled=True; IlfCommand=SLIN
;ENDFOLD
SLIN XP169 WITH $VEL = SVEL_CP(2.0, , LCPDAT169),$TOOL = STOOL2(FP169),$BASE = SBASE(FP169.BASE_NO),$IPO_MODE = SIPO_MODE(FP169.IPO_FRAME),$LOAD = SLOAD(FP169.TOOL_NO),$ACC = SACC_CP(LCPDAT169),$ORI_TYPE = SORI_TYP(LCPDAT169),$APO = SAPO(LCPDAT169),$JERK = SJERK(LCPDAT169),$COLLMON_TOL_PRO[1] = USE_CM_PRO_VALUES(0)
;ENDFOLD

;FOLD SLIN P170 Vel=2 m/s CPDAT170 Tool[4]:Microflown3D Base[2]:straight_sol;%{PE}
;FOLD Parameters ;%{h}
;Params IlfProvider=kukaroboter.basistech.inlineforms.movement.spline; Kuka.IsGlobalPoint=False; Kuka.PointName=P170; Kuka.BlendingEnabled=False; Kuka.MoveDataName=CPDAT170; Kuka.VelocityPath=2.000; Kuka.VelocityFieldEnabled=True; Kuka.ColDetectFieldEnabled=True; Kuka.CurrentCDSetIndex=0; Kuka.MovementParameterFieldEnabled=True; IlfCommand=SLIN
;ENDFOLD
SLIN XP170 WITH $VEL = SVEL_CP(2.0, , LCPDAT170),$TOOL = STOOL2(FP170),$BASE = SBASE(FP170.BASE_NO),$IPO_MODE = SIPO_MODE(FP170.IPO_FRAME),$LOAD = SLOAD(FP170.TOOL_NO),$ACC = SACC_CP(LCPDAT170),$ORI_TYPE = SORI_TYP(LCPDAT170),$APO = SAPO(LCPDAT170),$JERK = SJERK(LCPDAT170),$COLLMON_TOL_PRO[1] = USE_CM_PRO_VALUES(0)
;ENDFOLD

;FOLD SLIN P171 Vel=2 m/s CPDAT171 Tool[4]:Microflown3D Base[2]:straight_sol;%{PE}
;FOLD Parameters ;%{h}
;Params IlfProvider=kukaroboter.basistech.inlineforms.movement.spline; Kuka.IsGlobalPoint=False; Kuka.PointName=P171; Kuka.BlendingEnabled=False; Kuka.MoveDataName=CPDAT171; Kuka.VelocityPath=2.000; Kuka.VelocityFieldEnabled=True; Kuka.ColDetectFieldEnabled=True; Kuka.CurrentCDSetIndex=0; Kuka.MovementParameterFieldEnabled=True; IlfCommand=SLIN
;ENDFOLD
SLIN XP171 WITH $VEL = SVEL_CP(2.0, , LCPDAT171),$TOOL = STOOL2(FP171),$BASE = SBASE(FP171.BASE_NO),$IPO_MODE = SIPO_MODE(FP171.IPO_FRAME),$LOAD = SLOAD(FP171.TOOL_NO),$ACC = SACC_CP(LCPDAT171),$ORI_TYPE = SORI_TYP(LCPDAT171),$APO = SAPO(LCPDAT171),$JERK = SJERK(LCPDAT171),$COLLMON_TOL_PRO[1] = USE_CM_PRO_VALUES(0)
;ENDFOLD

;FOLD SLIN P172 Vel=2 m/s CPDAT172 Tool[4]:Microflown3D Base[2]:straight_sol;%{PE}
;FOLD Parameters ;%{h}
;Params IlfProvider=kukaroboter.basistech.inlineforms.movement.spline; Kuka.IsGlobalPoint=False; Kuka.PointName=P172; Kuka.BlendingEnabled=False; Kuka.MoveDataName=CPDAT172; Kuka.VelocityPath=2.000; Kuka.VelocityFieldEnabled=True; Kuka.ColDetectFieldEnabled=True; Kuka.CurrentCDSetIndex=0; Kuka.MovementParameterFieldEnabled=True; IlfCommand=SLIN
;ENDFOLD
SLIN XP172 WITH $VEL = SVEL_CP(2.0, , LCPDAT172),$TOOL = STOOL2(FP172),$BASE = SBASE(FP172.BASE_NO),$IPO_MODE = SIPO_MODE(FP172.IPO_FRAME),$LOAD = SLOAD(FP172.TOOL_NO),$ACC = SACC_CP(LCPDAT172),$ORI_TYPE = SORI_TYP(LCPDAT172),$APO = SAPO(LCPDAT172),$JERK = SJERK(LCPDAT172),$COLLMON_TOL_PRO[1] = USE_CM_PRO_VALUES(0)
;ENDFOLD

;FOLD SLIN P173 Vel=2 m/s CPDAT173 Tool[4]:Microflown3D Base[2]:straight_sol;%{PE}
;FOLD Parameters ;%{h}
;Params IlfProvider=kukaroboter.basistech.inlineforms.movement.spline; Kuka.IsGlobalPoint=False; Kuka.PointName=P173; Kuka.BlendingEnabled=False; Kuka.MoveDataName=CPDAT173; Kuka.VelocityPath=2.000; Kuka.VelocityFieldEnabled=True; Kuka.ColDetectFieldEnabled=True; Kuka.CurrentCDSetIndex=0; Kuka.MovementParameterFieldEnabled=True; IlfCommand=SLIN
;ENDFOLD
SLIN XP173 WITH $VEL = SVEL_CP(2.0, , LCPDAT173),$TOOL = STOOL2(FP173),$BASE = SBASE(FP173.BASE_NO),$IPO_MODE = SIPO_MODE(FP173.IPO_FRAME),$LOAD = SLOAD(FP173.TOOL_NO),$ACC = SACC_CP(LCPDAT173),$ORI_TYPE = SORI_TYP(LCPDAT173),$APO = SAPO(LCPDAT173),$JERK = SJERK(LCPDAT173),$COLLMON_TOL_PRO[1] = USE_CM_PRO_VALUES(0)
;ENDFOLD

;FOLD SLIN P174 Vel=2 m/s CPDAT174 Tool[4]:Microflown3D Base[2]:straight_sol;%{PE}
;FOLD Parameters ;%{h}
;Params IlfProvider=kukaroboter.basistech.inlineforms.movement.spline; Kuka.IsGlobalPoint=False; Kuka.PointName=P174; Kuka.BlendingEnabled=False; Kuka.MoveDataName=CPDAT174; Kuka.VelocityPath=2.000; Kuka.VelocityFieldEnabled=True; Kuka.ColDetectFieldEnabled=True; Kuka.CurrentCDSetIndex=0; Kuka.MovementParameterFieldEnabled=True; IlfCommand=SLIN
;ENDFOLD
SLIN XP174 WITH $VEL = SVEL_CP(2.0, , LCPDAT174),$TOOL = STOOL2(FP174),$BASE = SBASE(FP174.BASE_NO),$IPO_MODE = SIPO_MODE(FP174.IPO_FRAME),$LOAD = SLOAD(FP174.TOOL_NO),$ACC = SACC_CP(LCPDAT174),$ORI_TYPE = SORI_TYP(LCPDAT174),$APO = SAPO(LCPDAT174),$JERK = SJERK(LCPDAT174),$COLLMON_TOL_PRO[1] = USE_CM_PRO_VALUES(0)
;ENDFOLD

;FOLD SLIN P175 Vel=2 m/s CPDAT175 Tool[4]:Microflown3D Base[2]:straight_sol;%{PE}
;FOLD Parameters ;%{h}
;Params IlfProvider=kukaroboter.basistech.inlineforms.movement.spline; Kuka.IsGlobalPoint=False; Kuka.PointName=P175; Kuka.BlendingEnabled=False; Kuka.MoveDataName=CPDAT175; Kuka.VelocityPath=2.000; Kuka.VelocityFieldEnabled=True; Kuka.ColDetectFieldEnabled=True; Kuka.CurrentCDSetIndex=0; Kuka.MovementParameterFieldEnabled=True; IlfCommand=SLIN
;ENDFOLD
SLIN XP175 WITH $VEL = SVEL_CP(2.0, , LCPDAT175),$TOOL = STOOL2(FP175),$BASE = SBASE(FP175.BASE_NO),$IPO_MODE = SIPO_MODE(FP175.IPO_FRAME),$LOAD = SLOAD(FP175.TOOL_NO),$ACC = SACC_CP(LCPDAT175),$ORI_TYPE = SORI_TYP(LCPDAT175),$APO = SAPO(LCPDAT175),$JERK = SJERK(LCPDAT175),$COLLMON_TOL_PRO[1] = USE_CM_PRO_VALUES(0)
;ENDFOLD

;FOLD SLIN P176 Vel=2 m/s CPDAT176 Tool[4]:Microflown3D Base[2]:straight_sol;%{PE}
;FOLD Parameters ;%{h}
;Params IlfProvider=kukaroboter.basistech.inlineforms.movement.spline; Kuka.IsGlobalPoint=False; Kuka.PointName=P176; Kuka.BlendingEnabled=False; Kuka.MoveDataName=CPDAT176; Kuka.VelocityPath=2.000; Kuka.VelocityFieldEnabled=True; Kuka.ColDetectFieldEnabled=True; Kuka.CurrentCDSetIndex=0; Kuka.MovementParameterFieldEnabled=True; IlfCommand=SLIN
;ENDFOLD
SLIN XP176 WITH $VEL = SVEL_CP(2.0, , LCPDAT176),$TOOL = STOOL2(FP176),$BASE = SBASE(FP176.BASE_NO),$IPO_MODE = SIPO_MODE(FP176.IPO_FRAME),$LOAD = SLOAD(FP176.TOOL_NO),$ACC = SACC_CP(LCPDAT176),$ORI_TYPE = SORI_TYP(LCPDAT176),$APO = SAPO(LCPDAT176),$JERK = SJERK(LCPDAT176),$COLLMON_TOL_PRO[1] = USE_CM_PRO_VALUES(0)
;ENDFOLD

;FOLD SLIN P177 Vel=2 m/s CPDAT177 Tool[4]:Microflown3D Base[2]:straight_sol;%{PE}
;FOLD Parameters ;%{h}
;Params IlfProvider=kukaroboter.basistech.inlineforms.movement.spline; Kuka.IsGlobalPoint=False; Kuka.PointName=P177; Kuka.BlendingEnabled=False; Kuka.MoveDataName=CPDAT177; Kuka.VelocityPath=2.000; Kuka.VelocityFieldEnabled=True; Kuka.ColDetectFieldEnabled=True; Kuka.CurrentCDSetIndex=0; Kuka.MovementParameterFieldEnabled=True; IlfCommand=SLIN
;ENDFOLD
SLIN XP177 WITH $VEL = SVEL_CP(2.0, , LCPDAT177),$TOOL = STOOL2(FP177),$BASE = SBASE(FP177.BASE_NO),$IPO_MODE = SIPO_MODE(FP177.IPO_FRAME),$LOAD = SLOAD(FP177.TOOL_NO),$ACC = SACC_CP(LCPDAT177),$ORI_TYPE = SORI_TYP(LCPDAT177),$APO = SAPO(LCPDAT177),$JERK = SJERK(LCPDAT177),$COLLMON_TOL_PRO[1] = USE_CM_PRO_VALUES(0)
;ENDFOLD

;FOLD SLIN P178 Vel=2 m/s CPDAT178 Tool[4]:Microflown3D Base[2]:straight_sol;%{PE}
;FOLD Parameters ;%{h}
;Params IlfProvider=kukaroboter.basistech.inlineforms.movement.spline; Kuka.IsGlobalPoint=False; Kuka.PointName=P178; Kuka.BlendingEnabled=False; Kuka.MoveDataName=CPDAT178; Kuka.VelocityPath=2.000; Kuka.VelocityFieldEnabled=True; Kuka.ColDetectFieldEnabled=True; Kuka.CurrentCDSetIndex=0; Kuka.MovementParameterFieldEnabled=True; IlfCommand=SLIN
;ENDFOLD
SLIN XP178 WITH $VEL = SVEL_CP(2.0, , LCPDAT178),$TOOL = STOOL2(FP178),$BASE = SBASE(FP178.BASE_NO),$IPO_MODE = SIPO_MODE(FP178.IPO_FRAME),$LOAD = SLOAD(FP178.TOOL_NO),$ACC = SACC_CP(LCPDAT178),$ORI_TYPE = SORI_TYP(LCPDAT178),$APO = SAPO(LCPDAT178),$JERK = SJERK(LCPDAT178),$COLLMON_TOL_PRO[1] = USE_CM_PRO_VALUES(0)
;ENDFOLD

;FOLD SLIN P179 Vel=2 m/s CPDAT179 Tool[4]:Microflown3D Base[2]:straight_sol;%{PE}
;FOLD Parameters ;%{h}
;Params IlfProvider=kukaroboter.basistech.inlineforms.movement.spline; Kuka.IsGlobalPoint=False; Kuka.PointName=P179; Kuka.BlendingEnabled=False; Kuka.MoveDataName=CPDAT179; Kuka.VelocityPath=2.000; Kuka.VelocityFieldEnabled=True; Kuka.ColDetectFieldEnabled=True; Kuka.CurrentCDSetIndex=0; Kuka.MovementParameterFieldEnabled=True; IlfCommand=SLIN
;ENDFOLD
SLIN XP179 WITH $VEL = SVEL_CP(2.0, , LCPDAT179),$TOOL = STOOL2(FP179),$BASE = SBASE(FP179.BASE_NO),$IPO_MODE = SIPO_MODE(FP179.IPO_FRAME),$LOAD = SLOAD(FP179.TOOL_NO),$ACC = SACC_CP(LCPDAT179),$ORI_TYPE = SORI_TYP(LCPDAT179),$APO = SAPO(LCPDAT179),$JERK = SJERK(LCPDAT179),$COLLMON_TOL_PRO[1] = USE_CM_PRO_VALUES(0)
;ENDFOLD

;FOLD SLIN P180 Vel=2 m/s CPDAT180 Tool[4]:Microflown3D Base[2]:straight_sol;%{PE}
;FOLD Parameters ;%{h}
;Params IlfProvider=kukaroboter.basistech.inlineforms.movement.spline; Kuka.IsGlobalPoint=False; Kuka.PointName=P180; Kuka.BlendingEnabled=False; Kuka.MoveDataName=CPDAT180; Kuka.VelocityPath=2.000; Kuka.VelocityFieldEnabled=True; Kuka.ColDetectFieldEnabled=True; Kuka.CurrentCDSetIndex=0; Kuka.MovementParameterFieldEnabled=True; IlfCommand=SLIN
;ENDFOLD
SLIN XP180 WITH $VEL = SVEL_CP(2.0, , LCPDAT180),$TOOL = STOOL2(FP180),$BASE = SBASE(FP180.BASE_NO),$IPO_MODE = SIPO_MODE(FP180.IPO_FRAME),$LOAD = SLOAD(FP180.TOOL_NO),$ACC = SACC_CP(LCPDAT180),$ORI_TYPE = SORI_TYP(LCPDAT180),$APO = SAPO(LCPDAT180),$JERK = SJERK(LCPDAT180),$COLLMON_TOL_PRO[1] = USE_CM_PRO_VALUES(0)
;ENDFOLD

;FOLD SLIN P181 Vel=2 m/s CPDAT181 Tool[4]:Microflown3D Base[2]:straight_sol;%{PE}
;FOLD Parameters ;%{h}
;Params IlfProvider=kukaroboter.basistech.inlineforms.movement.spline; Kuka.IsGlobalPoint=False; Kuka.PointName=P181; Kuka.BlendingEnabled=False; Kuka.MoveDataName=CPDAT181; Kuka.VelocityPath=2.000; Kuka.VelocityFieldEnabled=True; Kuka.ColDetectFieldEnabled=True; Kuka.CurrentCDSetIndex=0; Kuka.MovementParameterFieldEnabled=True; IlfCommand=SLIN
;ENDFOLD
SLIN XP181 WITH $VEL = SVEL_CP(2.0, , LCPDAT181),$TOOL = STOOL2(FP181),$BASE = SBASE(FP181.BASE_NO),$IPO_MODE = SIPO_MODE(FP181.IPO_FRAME),$LOAD = SLOAD(FP181.TOOL_NO),$ACC = SACC_CP(LCPDAT181),$ORI_TYPE = SORI_TYP(LCPDAT181),$APO = SAPO(LCPDAT181),$JERK = SJERK(LCPDAT181),$COLLMON_TOL_PRO[1] = USE_CM_PRO_VALUES(0)
;ENDFOLD

;FOLD SLIN P182 Vel=2 m/s CPDAT182 Tool[4]:Microflown3D Base[2]:straight_sol;%{PE}
;FOLD Parameters ;%{h}
;Params IlfProvider=kukaroboter.basistech.inlineforms.movement.spline; Kuka.IsGlobalPoint=False; Kuka.PointName=P182; Kuka.BlendingEnabled=False; Kuka.MoveDataName=CPDAT182; Kuka.VelocityPath=2.000; Kuka.VelocityFieldEnabled=True; Kuka.ColDetectFieldEnabled=True; Kuka.CurrentCDSetIndex=0; Kuka.MovementParameterFieldEnabled=True; IlfCommand=SLIN
;ENDFOLD
SLIN XP182 WITH $VEL = SVEL_CP(2.0, , LCPDAT182),$TOOL = STOOL2(FP182),$BASE = SBASE(FP182.BASE_NO),$IPO_MODE = SIPO_MODE(FP182.IPO_FRAME),$LOAD = SLOAD(FP182.TOOL_NO),$ACC = SACC_CP(LCPDAT182),$ORI_TYPE = SORI_TYP(LCPDAT182),$APO = SAPO(LCPDAT182),$JERK = SJERK(LCPDAT182),$COLLMON_TOL_PRO[1] = USE_CM_PRO_VALUES(0)
;ENDFOLD

;FOLD SLIN P183 Vel=2 m/s CPDAT183 Tool[4]:Microflown3D Base[2]:straight_sol;%{PE}
;FOLD Parameters ;%{h}
;Params IlfProvider=kukaroboter.basistech.inlineforms.movement.spline; Kuka.IsGlobalPoint=False; Kuka.PointName=P183; Kuka.BlendingEnabled=False; Kuka.MoveDataName=CPDAT183; Kuka.VelocityPath=2.000; Kuka.VelocityFieldEnabled=True; Kuka.ColDetectFieldEnabled=True; Kuka.CurrentCDSetIndex=0; Kuka.MovementParameterFieldEnabled=True; IlfCommand=SLIN
;ENDFOLD
SLIN XP183 WITH $VEL = SVEL_CP(2.0, , LCPDAT183),$TOOL = STOOL2(FP183),$BASE = SBASE(FP183.BASE_NO),$IPO_MODE = SIPO_MODE(FP183.IPO_FRAME),$LOAD = SLOAD(FP183.TOOL_NO),$ACC = SACC_CP(LCPDAT183),$ORI_TYPE = SORI_TYP(LCPDAT183),$APO = SAPO(LCPDAT183),$JERK = SJERK(LCPDAT183),$COLLMON_TOL_PRO[1] = USE_CM_PRO_VALUES(0)
;ENDFOLD

;FOLD SLIN P184 Vel=2 m/s CPDAT184 Tool[4]:Microflown3D Base[2]:straight_sol;%{PE}
;FOLD Parameters ;%{h}
;Params IlfProvider=kukaroboter.basistech.inlineforms.movement.spline; Kuka.IsGlobalPoint=False; Kuka.PointName=P184; Kuka.BlendingEnabled=False; Kuka.MoveDataName=CPDAT184; Kuka.VelocityPath=2.000; Kuka.VelocityFieldEnabled=True; Kuka.ColDetectFieldEnabled=True; Kuka.CurrentCDSetIndex=0; Kuka.MovementParameterFieldEnabled=True; IlfCommand=SLIN
;ENDFOLD
SLIN XP184 WITH $VEL = SVEL_CP(2.0, , LCPDAT184),$TOOL = STOOL2(FP184),$BASE = SBASE(FP184.BASE_NO),$IPO_MODE = SIPO_MODE(FP184.IPO_FRAME),$LOAD = SLOAD(FP184.TOOL_NO),$ACC = SACC_CP(LCPDAT184),$ORI_TYPE = SORI_TYP(LCPDAT184),$APO = SAPO(LCPDAT184),$JERK = SJERK(LCPDAT184),$COLLMON_TOL_PRO[1] = USE_CM_PRO_VALUES(0)
;ENDFOLD

;FOLD SLIN P185 Vel=2 m/s CPDAT185 Tool[4]:Microflown3D Base[2]:straight_sol;%{PE}
;FOLD Parameters ;%{h}
;Params IlfProvider=kukaroboter.basistech.inlineforms.movement.spline; Kuka.IsGlobalPoint=False; Kuka.PointName=P185; Kuka.BlendingEnabled=False; Kuka.MoveDataName=CPDAT185; Kuka.VelocityPath=2.000; Kuka.VelocityFieldEnabled=True; Kuka.ColDetectFieldEnabled=True; Kuka.CurrentCDSetIndex=0; Kuka.MovementParameterFieldEnabled=True; IlfCommand=SLIN
;ENDFOLD
SLIN XP185 WITH $VEL = SVEL_CP(2.0, , LCPDAT185),$TOOL = STOOL2(FP185),$BASE = SBASE(FP185.BASE_NO),$IPO_MODE = SIPO_MODE(FP185.IPO_FRAME),$LOAD = SLOAD(FP185.TOOL_NO),$ACC = SACC_CP(LCPDAT185),$ORI_TYPE = SORI_TYP(LCPDAT185),$APO = SAPO(LCPDAT185),$JERK = SJERK(LCPDAT185),$COLLMON_TOL_PRO[1] = USE_CM_PRO_VALUES(0)
;ENDFOLD

;FOLD SLIN P186 Vel=2 m/s CPDAT186 Tool[4]:Microflown3D Base[2]:straight_sol;%{PE}
;FOLD Parameters ;%{h}
;Params IlfProvider=kukaroboter.basistech.inlineforms.movement.spline; Kuka.IsGlobalPoint=False; Kuka.PointName=P186; Kuka.BlendingEnabled=False; Kuka.MoveDataName=CPDAT186; Kuka.VelocityPath=2.000; Kuka.VelocityFieldEnabled=True; Kuka.ColDetectFieldEnabled=True; Kuka.CurrentCDSetIndex=0; Kuka.MovementParameterFieldEnabled=True; IlfCommand=SLIN
;ENDFOLD
SLIN XP186 WITH $VEL = SVEL_CP(2.0, , LCPDAT186),$TOOL = STOOL2(FP186),$BASE = SBASE(FP186.BASE_NO),$IPO_MODE = SIPO_MODE(FP186.IPO_FRAME),$LOAD = SLOAD(FP186.TOOL_NO),$ACC = SACC_CP(LCPDAT186),$ORI_TYPE = SORI_TYP(LCPDAT186),$APO = SAPO(LCPDAT186),$JERK = SJERK(LCPDAT186),$COLLMON_TOL_PRO[1] = USE_CM_PRO_VALUES(0)
;ENDFOLD

;FOLD SLIN P187 Vel=2 m/s CPDAT187 Tool[4]:Microflown3D Base[2]:straight_sol;%{PE}
;FOLD Parameters ;%{h}
;Params IlfProvider=kukaroboter.basistech.inlineforms.movement.spline; Kuka.IsGlobalPoint=False; Kuka.PointName=P187; Kuka.BlendingEnabled=False; Kuka.MoveDataName=CPDAT187; Kuka.VelocityPath=2.000; Kuka.VelocityFieldEnabled=True; Kuka.ColDetectFieldEnabled=True; Kuka.CurrentCDSetIndex=0; Kuka.MovementParameterFieldEnabled=True; IlfCommand=SLIN
;ENDFOLD
SLIN XP187 WITH $VEL = SVEL_CP(2.0, , LCPDAT187),$TOOL = STOOL2(FP187),$BASE = SBASE(FP187.BASE_NO),$IPO_MODE = SIPO_MODE(FP187.IPO_FRAME),$LOAD = SLOAD(FP187.TOOL_NO),$ACC = SACC_CP(LCPDAT187),$ORI_TYPE = SORI_TYP(LCPDAT187),$APO = SAPO(LCPDAT187),$JERK = SJERK(LCPDAT187),$COLLMON_TOL_PRO[1] = USE_CM_PRO_VALUES(0)
;ENDFOLD

;FOLD SLIN P188 Vel=2 m/s CPDAT188 Tool[4]:Microflown3D Base[2]:straight_sol;%{PE}
;FOLD Parameters ;%{h}
;Params IlfProvider=kukaroboter.basistech.inlineforms.movement.spline; Kuka.IsGlobalPoint=False; Kuka.PointName=P188; Kuka.BlendingEnabled=False; Kuka.MoveDataName=CPDAT188; Kuka.VelocityPath=2.000; Kuka.VelocityFieldEnabled=True; Kuka.ColDetectFieldEnabled=True; Kuka.CurrentCDSetIndex=0; Kuka.MovementParameterFieldEnabled=True; IlfCommand=SLIN
;ENDFOLD
SLIN XP188 WITH $VEL = SVEL_CP(2.0, , LCPDAT188),$TOOL = STOOL2(FP188),$BASE = SBASE(FP188.BASE_NO),$IPO_MODE = SIPO_MODE(FP188.IPO_FRAME),$LOAD = SLOAD(FP188.TOOL_NO),$ACC = SACC_CP(LCPDAT188),$ORI_TYPE = SORI_TYP(LCPDAT188),$APO = SAPO(LCPDAT188),$JERK = SJERK(LCPDAT188),$COLLMON_TOL_PRO[1] = USE_CM_PRO_VALUES(0)
;ENDFOLD

;FOLD SLIN P189 Vel=2 m/s CPDAT189 Tool[4]:Microflown3D Base[2]:straight_sol;%{PE}
;FOLD Parameters ;%{h}
;Params IlfProvider=kukaroboter.basistech.inlineforms.movement.spline; Kuka.IsGlobalPoint=False; Kuka.PointName=P189; Kuka.BlendingEnabled=False; Kuka.MoveDataName=CPDAT189; Kuka.VelocityPath=2.000; Kuka.VelocityFieldEnabled=True; Kuka.ColDetectFieldEnabled=True; Kuka.CurrentCDSetIndex=0; Kuka.MovementParameterFieldEnabled=True; IlfCommand=SLIN
;ENDFOLD
SLIN XP189 WITH $VEL = SVEL_CP(2.0, , LCPDAT189),$TOOL = STOOL2(FP189),$BASE = SBASE(FP189.BASE_NO),$IPO_MODE = SIPO_MODE(FP189.IPO_FRAME),$LOAD = SLOAD(FP189.TOOL_NO),$ACC = SACC_CP(LCPDAT189),$ORI_TYPE = SORI_TYP(LCPDAT189),$APO = SAPO(LCPDAT189),$JERK = SJERK(LCPDAT189),$COLLMON_TOL_PRO[1] = USE_CM_PRO_VALUES(0)
;ENDFOLD

;FOLD SLIN P190 Vel=2 m/s CPDAT190 Tool[4]:Microflown3D Base[2]:straight_sol;%{PE}
;FOLD Parameters ;%{h}
;Params IlfProvider=kukaroboter.basistech.inlineforms.movement.spline; Kuka.IsGlobalPoint=False; Kuka.PointName=P190; Kuka.BlendingEnabled=False; Kuka.MoveDataName=CPDAT190; Kuka.VelocityPath=2.000; Kuka.VelocityFieldEnabled=True; Kuka.ColDetectFieldEnabled=True; Kuka.CurrentCDSetIndex=0; Kuka.MovementParameterFieldEnabled=True; IlfCommand=SLIN
;ENDFOLD
SLIN XP190 WITH $VEL = SVEL_CP(2.0, , LCPDAT190),$TOOL = STOOL2(FP190),$BASE = SBASE(FP190.BASE_NO),$IPO_MODE = SIPO_MODE(FP190.IPO_FRAME),$LOAD = SLOAD(FP190.TOOL_NO),$ACC = SACC_CP(LCPDAT190),$ORI_TYPE = SORI_TYP(LCPDAT190),$APO = SAPO(LCPDAT190),$JERK = SJERK(LCPDAT190),$COLLMON_TOL_PRO[1] = USE_CM_PRO_VALUES(0)
;ENDFOLD

;FOLD SLIN P191 Vel=2 m/s CPDAT191 Tool[4]:Microflown3D Base[2]:straight_sol;%{PE}
;FOLD Parameters ;%{h}
;Params IlfProvider=kukaroboter.basistech.inlineforms.movement.spline; Kuka.IsGlobalPoint=False; Kuka.PointName=P191; Kuka.BlendingEnabled=False; Kuka.MoveDataName=CPDAT191; Kuka.VelocityPath=2.000; Kuka.VelocityFieldEnabled=True; Kuka.ColDetectFieldEnabled=True; Kuka.CurrentCDSetIndex=0; Kuka.MovementParameterFieldEnabled=True; IlfCommand=SLIN
;ENDFOLD
SLIN XP191 WITH $VEL = SVEL_CP(2.0, , LCPDAT191),$TOOL = STOOL2(FP191),$BASE = SBASE(FP191.BASE_NO),$IPO_MODE = SIPO_MODE(FP191.IPO_FRAME),$LOAD = SLOAD(FP191.TOOL_NO),$ACC = SACC_CP(LCPDAT191),$ORI_TYPE = SORI_TYP(LCPDAT191),$APO = SAPO(LCPDAT191),$JERK = SJERK(LCPDAT191),$COLLMON_TOL_PRO[1] = USE_CM_PRO_VALUES(0)
;ENDFOLD

;FOLD SLIN P192 Vel=2 m/s CPDAT192 Tool[4]:Microflown3D Base[2]:straight_sol;%{PE}
;FOLD Parameters ;%{h}
;Params IlfProvider=kukaroboter.basistech.inlineforms.movement.spline; Kuka.IsGlobalPoint=False; Kuka.PointName=P192; Kuka.BlendingEnabled=False; Kuka.MoveDataName=CPDAT192; Kuka.VelocityPath=2.000; Kuka.VelocityFieldEnabled=True; Kuka.ColDetectFieldEnabled=True; Kuka.CurrentCDSetIndex=0; Kuka.MovementParameterFieldEnabled=True; IlfCommand=SLIN
;ENDFOLD
SLIN XP192 WITH $VEL = SVEL_CP(2.0, , LCPDAT192),$TOOL = STOOL2(FP192),$BASE = SBASE(FP192.BASE_NO),$IPO_MODE = SIPO_MODE(FP192.IPO_FRAME),$LOAD = SLOAD(FP192.TOOL_NO),$ACC = SACC_CP(LCPDAT192),$ORI_TYPE = SORI_TYP(LCPDAT192),$APO = SAPO(LCPDAT192),$JERK = SJERK(LCPDAT192),$COLLMON_TOL_PRO[1] = USE_CM_PRO_VALUES(0)
;ENDFOLD

;FOLD SLIN P193 Vel=2 m/s CPDAT193 Tool[4]:Microflown3D Base[2]:straight_sol;%{PE}
;FOLD Parameters ;%{h}
;Params IlfProvider=kukaroboter.basistech.inlineforms.movement.spline; Kuka.IsGlobalPoint=False; Kuka.PointName=P193; Kuka.BlendingEnabled=False; Kuka.MoveDataName=CPDAT193; Kuka.VelocityPath=2.000; Kuka.VelocityFieldEnabled=True; Kuka.ColDetectFieldEnabled=True; Kuka.CurrentCDSetIndex=0; Kuka.MovementParameterFieldEnabled=True; IlfCommand=SLIN
;ENDFOLD
SLIN XP193 WITH $VEL = SVEL_CP(2.0, , LCPDAT193),$TOOL = STOOL2(FP193),$BASE = SBASE(FP193.BASE_NO),$IPO_MODE = SIPO_MODE(FP193.IPO_FRAME),$LOAD = SLOAD(FP193.TOOL_NO),$ACC = SACC_CP(LCPDAT193),$ORI_TYPE = SORI_TYP(LCPDAT193),$APO = SAPO(LCPDAT193),$JERK = SJERK(LCPDAT193),$COLLMON_TOL_PRO[1] = USE_CM_PRO_VALUES(0)
;ENDFOLD

;FOLD SLIN P194 Vel=2 m/s CPDAT194 Tool[4]:Microflown3D Base[2]:straight_sol;%{PE}
;FOLD Parameters ;%{h}
;Params IlfProvider=kukaroboter.basistech.inlineforms.movement.spline; Kuka.IsGlobalPoint=False; Kuka.PointName=P194; Kuka.BlendingEnabled=False; Kuka.MoveDataName=CPDAT194; Kuka.VelocityPath=2.000; Kuka.VelocityFieldEnabled=True; Kuka.ColDetectFieldEnabled=True; Kuka.CurrentCDSetIndex=0; Kuka.MovementParameterFieldEnabled=True; IlfCommand=SLIN
;ENDFOLD
SLIN XP194 WITH $VEL = SVEL_CP(2.0, , LCPDAT194),$TOOL = STOOL2(FP194),$BASE = SBASE(FP194.BASE_NO),$IPO_MODE = SIPO_MODE(FP194.IPO_FRAME),$LOAD = SLOAD(FP194.TOOL_NO),$ACC = SACC_CP(LCPDAT194),$ORI_TYPE = SORI_TYP(LCPDAT194),$APO = SAPO(LCPDAT194),$JERK = SJERK(LCPDAT194),$COLLMON_TOL_PRO[1] = USE_CM_PRO_VALUES(0)
;ENDFOLD

;FOLD SLIN P195 Vel=2 m/s CPDAT195 Tool[4]:Microflown3D Base[2]:straight_sol;%{PE}
;FOLD Parameters ;%{h}
;Params IlfProvider=kukaroboter.basistech.inlineforms.movement.spline; Kuka.IsGlobalPoint=False; Kuka.PointName=P195; Kuka.BlendingEnabled=False; Kuka.MoveDataName=CPDAT195; Kuka.VelocityPath=2.000; Kuka.VelocityFieldEnabled=True; Kuka.ColDetectFieldEnabled=True; Kuka.CurrentCDSetIndex=0; Kuka.MovementParameterFieldEnabled=True; IlfCommand=SLIN
;ENDFOLD
SLIN XP195 WITH $VEL = SVEL_CP(2.0, , LCPDAT195),$TOOL = STOOL2(FP195),$BASE = SBASE(FP195.BASE_NO),$IPO_MODE = SIPO_MODE(FP195.IPO_FRAME),$LOAD = SLOAD(FP195.TOOL_NO),$ACC = SACC_CP(LCPDAT195),$ORI_TYPE = SORI_TYP(LCPDAT195),$APO = SAPO(LCPDAT195),$JERK = SJERK(LCPDAT195),$COLLMON_TOL_PRO[1] = USE_CM_PRO_VALUES(0)
;ENDFOLD

;FOLD SLIN P196 Vel=2 m/s CPDAT196 Tool[4]:Microflown3D Base[2]:straight_sol;%{PE}
;FOLD Parameters ;%{h}
;Params IlfProvider=kukaroboter.basistech.inlineforms.movement.spline; Kuka.IsGlobalPoint=False; Kuka.PointName=P196; Kuka.BlendingEnabled=False; Kuka.MoveDataName=CPDAT196; Kuka.VelocityPath=2.000; Kuka.VelocityFieldEnabled=True; Kuka.ColDetectFieldEnabled=True; Kuka.CurrentCDSetIndex=0; Kuka.MovementParameterFieldEnabled=True; IlfCommand=SLIN
;ENDFOLD
SLIN XP196 WITH $VEL = SVEL_CP(2.0, , LCPDAT196),$TOOL = STOOL2(FP196),$BASE = SBASE(FP196.BASE_NO),$IPO_MODE = SIPO_MODE(FP196.IPO_FRAME),$LOAD = SLOAD(FP196.TOOL_NO),$ACC = SACC_CP(LCPDAT196),$ORI_TYPE = SORI_TYP(LCPDAT196),$APO = SAPO(LCPDAT196),$JERK = SJERK(LCPDAT196),$COLLMON_TOL_PRO[1] = USE_CM_PRO_VALUES(0)
;ENDFOLD

;FOLD SLIN P197 Vel=2 m/s CPDAT197 Tool[4]:Microflown3D Base[2]:straight_sol;%{PE}
;FOLD Parameters ;%{h}
;Params IlfProvider=kukaroboter.basistech.inlineforms.movement.spline; Kuka.IsGlobalPoint=False; Kuka.PointName=P197; Kuka.BlendingEnabled=False; Kuka.MoveDataName=CPDAT197; Kuka.VelocityPath=2.000; Kuka.VelocityFieldEnabled=True; Kuka.ColDetectFieldEnabled=True; Kuka.CurrentCDSetIndex=0; Kuka.MovementParameterFieldEnabled=True; IlfCommand=SLIN
;ENDFOLD
SLIN XP197 WITH $VEL = SVEL_CP(2.0, , LCPDAT197),$TOOL = STOOL2(FP197),$BASE = SBASE(FP197.BASE_NO),$IPO_MODE = SIPO_MODE(FP197.IPO_FRAME),$LOAD = SLOAD(FP197.TOOL_NO),$ACC = SACC_CP(LCPDAT197),$ORI_TYPE = SORI_TYP(LCPDAT197),$APO = SAPO(LCPDAT197),$JERK = SJERK(LCPDAT197),$COLLMON_TOL_PRO[1] = USE_CM_PRO_VALUES(0)
;ENDFOLD

;FOLD SLIN P198 Vel=2 m/s CPDAT198 Tool[4]:Microflown3D Base[2]:straight_sol;%{PE}
;FOLD Parameters ;%{h}
;Params IlfProvider=kukaroboter.basistech.inlineforms.movement.spline; Kuka.IsGlobalPoint=False; Kuka.PointName=P198; Kuka.BlendingEnabled=False; Kuka.MoveDataName=CPDAT198; Kuka.VelocityPath=2.000; Kuka.VelocityFieldEnabled=True; Kuka.ColDetectFieldEnabled=True; Kuka.CurrentCDSetIndex=0; Kuka.MovementParameterFieldEnabled=True; IlfCommand=SLIN
;ENDFOLD
SLIN XP198 WITH $VEL = SVEL_CP(2.0, , LCPDAT198),$TOOL = STOOL2(FP198),$BASE = SBASE(FP198.BASE_NO),$IPO_MODE = SIPO_MODE(FP198.IPO_FRAME),$LOAD = SLOAD(FP198.TOOL_NO),$ACC = SACC_CP(LCPDAT198),$ORI_TYPE = SORI_TYP(LCPDAT198),$APO = SAPO(LCPDAT198),$JERK = SJERK(LCPDAT198),$COLLMON_TOL_PRO[1] = USE_CM_PRO_VALUES(0)
;ENDFOLD

;FOLD SLIN P199 Vel=2 m/s CPDAT199 Tool[4]:Microflown3D Base[2]:straight_sol;%{PE}
;FOLD Parameters ;%{h}
;Params IlfProvider=kukaroboter.basistech.inlineforms.movement.spline; Kuka.IsGlobalPoint=False; Kuka.PointName=P199; Kuka.BlendingEnabled=False; Kuka.MoveDataName=CPDAT199; Kuka.VelocityPath=2.000; Kuka.VelocityFieldEnabled=True; Kuka.ColDetectFieldEnabled=True; Kuka.CurrentCDSetIndex=0; Kuka.MovementParameterFieldEnabled=True; IlfCommand=SLIN
;ENDFOLD
SLIN XP199 WITH $VEL = SVEL_CP(2.0, , LCPDAT199),$TOOL = STOOL2(FP199),$BASE = SBASE(FP199.BASE_NO),$IPO_MODE = SIPO_MODE(FP199.IPO_FRAME),$LOAD = SLOAD(FP199.TOOL_NO),$ACC = SACC_CP(LCPDAT199),$ORI_TYPE = SORI_TYP(LCPDAT199),$APO = SAPO(LCPDAT199),$JERK = SJERK(LCPDAT199),$COLLMON_TOL_PRO[1] = USE_CM_PRO_VALUES(0)
;ENDFOLD

;FOLD SLIN P200 Vel=2 m/s CPDAT200 Tool[4]:Microflown3D Base[2]:straight_sol;%{PE}
;FOLD Parameters ;%{h}
;Params IlfProvider=kukaroboter.basistech.inlineforms.movement.spline; Kuka.IsGlobalPoint=False; Kuka.PointName=P200; Kuka.BlendingEnabled=False; Kuka.MoveDataName=CPDAT200; Kuka.VelocityPath=2.000; Kuka.VelocityFieldEnabled=True; Kuka.ColDetectFieldEnabled=True; Kuka.CurrentCDSetIndex=0; Kuka.MovementParameterFieldEnabled=True; IlfCommand=SLIN
;ENDFOLD
SLIN XP200 WITH $VEL = SVEL_CP(2.0, , LCPDAT200),$TOOL = STOOL2(FP200),$BASE = SBASE(FP200.BASE_NO),$IPO_MODE = SIPO_MODE(FP200.IPO_FRAME),$LOAD = SLOAD(FP200.TOOL_NO),$ACC = SACC_CP(LCPDAT200),$ORI_TYPE = SORI_TYP(LCPDAT200),$APO = SAPO(LCPDAT200),$JERK = SJERK(LCPDAT200),$COLLMON_TOL_PRO[1] = USE_CM_PRO_VALUES(0)
;ENDFOLD

;FOLD SLIN P201 Vel=2 m/s CPDAT201 Tool[4]:Microflown3D Base[2]:straight_sol;%{PE}
;FOLD Parameters ;%{h}
;Params IlfProvider=kukaroboter.basistech.inlineforms.movement.spline; Kuka.IsGlobalPoint=False; Kuka.PointName=P201; Kuka.BlendingEnabled=False; Kuka.MoveDataName=CPDAT201; Kuka.VelocityPath=2.000; Kuka.VelocityFieldEnabled=True; Kuka.ColDetectFieldEnabled=True; Kuka.CurrentCDSetIndex=0; Kuka.MovementParameterFieldEnabled=True; IlfCommand=SLIN
;ENDFOLD
SLIN XP201 WITH $VEL = SVEL_CP(2.0, , LCPDAT201),$TOOL = STOOL2(FP201),$BASE = SBASE(FP201.BASE_NO),$IPO_MODE = SIPO_MODE(FP201.IPO_FRAME),$LOAD = SLOAD(FP201.TOOL_NO),$ACC = SACC_CP(LCPDAT201),$ORI_TYPE = SORI_TYP(LCPDAT201),$APO = SAPO(LCPDAT201),$JERK = SJERK(LCPDAT201),$COLLMON_TOL_PRO[1] = USE_CM_PRO_VALUES(0)
;ENDFOLD

;FOLD SLIN P202 Vel=2 m/s CPDAT202 Tool[4]:Microflown3D Base[2]:straight_sol;%{PE}
;FOLD Parameters ;%{h}
;Params IlfProvider=kukaroboter.basistech.inlineforms.movement.spline; Kuka.IsGlobalPoint=False; Kuka.PointName=P202; Kuka.BlendingEnabled=False; Kuka.MoveDataName=CPDAT202; Kuka.VelocityPath=2.000; Kuka.VelocityFieldEnabled=True; Kuka.ColDetectFieldEnabled=True; Kuka.CurrentCDSetIndex=0; Kuka.MovementParameterFieldEnabled=True; IlfCommand=SLIN
;ENDFOLD
SLIN XP202 WITH $VEL = SVEL_CP(2.0, , LCPDAT202),$TOOL = STOOL2(FP202),$BASE = SBASE(FP202.BASE_NO),$IPO_MODE = SIPO_MODE(FP202.IPO_FRAME),$LOAD = SLOAD(FP202.TOOL_NO),$ACC = SACC_CP(LCPDAT202),$ORI_TYPE = SORI_TYP(LCPDAT202),$APO = SAPO(LCPDAT202),$JERK = SJERK(LCPDAT202),$COLLMON_TOL_PRO[1] = USE_CM_PRO_VALUES(0)
;ENDFOLD

;FOLD SLIN P203 Vel=1 m/s CPDAT203 Tool[4]:Microflown3D Base[2]:straight_sol;%{PE}
;FOLD Parameters ;%{h}
;Params IlfProvider=kukaroboter.basistech.inlineforms.movement.spline; Kuka.IsGlobalPoint=False; Kuka.PointName=P203; Kuka.BlendingEnabled=False; Kuka.MoveDataName=CPDAT203; Kuka.VelocityPath=1.000; Kuka.VelocityFieldEnabled=True; Kuka.ColDetectFieldEnabled=True; Kuka.CurrentCDSetIndex=0; Kuka.MovementParameterFieldEnabled=True; IlfCommand=SLIN
;ENDFOLD
SLIN XP203 WITH $VEL = SVEL_CP(2.0, , LCPDAT203),$TOOL = STOOL2(FP203),$BASE = SBASE(FP203.BASE_NO),$IPO_MODE = SIPO_MODE(FP203.IPO_FRAME),$LOAD = SLOAD(FP203.TOOL_NO),$ACC = SACC_CP(LCPDAT203),$ORI_TYPE = SORI_TYP(LCPDAT203),$APO = SAPO(LCPDAT203),$JERK = SJERK(LCPDAT203),$COLLMON_TOL_PRO[1] = USE_CM_PRO_VALUES(0)
;ENDFOLD

;FOLD SLIN P204 Vel=1 m/s CPDAT204 Tool[4]:Microflown3D Base[2]:straight_sol;%{PE}
;FOLD Parameters ;%{h}
;Params IlfProvider=kukaroboter.basistech.inlineforms.movement.spline; Kuka.IsGlobalPoint=False; Kuka.PointName=P204; Kuka.BlendingEnabled=False; Kuka.MoveDataName=CPDAT204; Kuka.VelocityPath=1.000; Kuka.VelocityFieldEnabled=True; Kuka.ColDetectFieldEnabled=True; Kuka.CurrentCDSetIndex=0; Kuka.MovementParameterFieldEnabled=True; IlfCommand=SLIN
;ENDFOLD
SLIN XP204 WITH $VEL = SVEL_CP(2.0, , LCPDAT204),$TOOL = STOOL2(FP204),$BASE = SBASE(FP204.BASE_NO),$IPO_MODE = SIPO_MODE(FP204.IPO_FRAME),$LOAD = SLOAD(FP204.TOOL_NO),$ACC = SACC_CP(LCPDAT204),$ORI_TYPE = SORI_TYP(LCPDAT204),$APO = SAPO(LCPDAT204),$JERK = SJERK(LCPDAT204),$COLLMON_TOL_PRO[1] = USE_CM_PRO_VALUES(0)
;ENDFOLD

;FOLD SLIN P205 Vel=2 m/s CPDAT205 Tool[4]:Microflown3D Base[2]:straight_sol;%{PE}
;FOLD Parameters ;%{h}
;Params IlfProvider=kukaroboter.basistech.inlineforms.movement.spline; Kuka.IsGlobalPoint=False; Kuka.PointName=P205; Kuka.BlendingEnabled=False; Kuka.MoveDataName=CPDAT205; Kuka.VelocityPath=2.000; Kuka.VelocityFieldEnabled=True; Kuka.ColDetectFieldEnabled=True; Kuka.CurrentCDSetIndex=0; Kuka.MovementParameterFieldEnabled=True; IlfCommand=SLIN
;ENDFOLD
SLIN XP205 WITH $VEL = SVEL_CP(2.0, , LCPDAT205),$TOOL = STOOL2(FP205),$BASE = SBASE(FP205.BASE_NO),$IPO_MODE = SIPO_MODE(FP205.IPO_FRAME),$LOAD = SLOAD(FP205.TOOL_NO),$ACC = SACC_CP(LCPDAT205),$ORI_TYPE = SORI_TYP(LCPDAT205),$APO = SAPO(LCPDAT205),$JERK = SJERK(LCPDAT205),$COLLMON_TOL_PRO[1] = USE_CM_PRO_VALUES(0)
;ENDFOLD

;FOLD SLIN P206 Vel=2 m/s CPDAT206 Tool[4]:Microflown3D Base[2]:straight_sol;%{PE}
;FOLD Parameters ;%{h}
;Params IlfProvider=kukaroboter.basistech.inlineforms.movement.spline; Kuka.IsGlobalPoint=False; Kuka.PointName=P206; Kuka.BlendingEnabled=False; Kuka.MoveDataName=CPDAT206; Kuka.VelocityPath=2.000; Kuka.VelocityFieldEnabled=True; Kuka.ColDetectFieldEnabled=True; Kuka.CurrentCDSetIndex=0; Kuka.MovementParameterFieldEnabled=True; IlfCommand=SLIN
;ENDFOLD
SLIN XP206 WITH $VEL = SVEL_CP(2.0, , LCPDAT206),$TOOL = STOOL2(FP206),$BASE = SBASE(FP206.BASE_NO),$IPO_MODE = SIPO_MODE(FP206.IPO_FRAME),$LOAD = SLOAD(FP206.TOOL_NO),$ACC = SACC_CP(LCPDAT206),$ORI_TYPE = SORI_TYP(LCPDAT206),$APO = SAPO(LCPDAT206),$JERK = SJERK(LCPDAT206),$COLLMON_TOL_PRO[1] = USE_CM_PRO_VALUES(0)
;ENDFOLD

;FOLD SLIN P207 Vel=2 m/s CPDAT207 Tool[4]:Microflown3D Base[2]:straight_sol;%{PE}
;FOLD Parameters ;%{h}
;Params IlfProvider=kukaroboter.basistech.inlineforms.movement.spline; Kuka.IsGlobalPoint=False; Kuka.PointName=P207; Kuka.BlendingEnabled=False; Kuka.MoveDataName=CPDAT207; Kuka.VelocityPath=2.000; Kuka.VelocityFieldEnabled=True; Kuka.ColDetectFieldEnabled=True; Kuka.CurrentCDSetIndex=0; Kuka.MovementParameterFieldEnabled=True; IlfCommand=SLIN
;ENDFOLD
SLIN XP207 WITH $VEL = SVEL_CP(2.0, , LCPDAT207),$TOOL = STOOL2(FP207),$BASE = SBASE(FP207.BASE_NO),$IPO_MODE = SIPO_MODE(FP207.IPO_FRAME),$LOAD = SLOAD(FP207.TOOL_NO),$ACC = SACC_CP(LCPDAT207),$ORI_TYPE = SORI_TYP(LCPDAT207),$APO = SAPO(LCPDAT207),$JERK = SJERK(LCPDAT207),$COLLMON_TOL_PRO[1] = USE_CM_PRO_VALUES(0)
;ENDFOLD

;FOLD SLIN P208 Vel=2 m/s CPDAT208 Tool[4]:Microflown3D Base[2]:straight_sol;%{PE}
;FOLD Parameters ;%{h}
;Params IlfProvider=kukaroboter.basistech.inlineforms.movement.spline; Kuka.IsGlobalPoint=False; Kuka.PointName=P208; Kuka.BlendingEnabled=False; Kuka.MoveDataName=CPDAT208; Kuka.VelocityPath=2.000; Kuka.VelocityFieldEnabled=True; Kuka.ColDetectFieldEnabled=True; Kuka.CurrentCDSetIndex=0; Kuka.MovementParameterFieldEnabled=True; IlfCommand=SLIN
;ENDFOLD
SLIN XP208 WITH $VEL = SVEL_CP(2.0, , LCPDAT208),$TOOL = STOOL2(FP208),$BASE = SBASE(FP208.BASE_NO),$IPO_MODE = SIPO_MODE(FP208.IPO_FRAME),$LOAD = SLOAD(FP208.TOOL_NO),$ACC = SACC_CP(LCPDAT208),$ORI_TYPE = SORI_TYP(LCPDAT208),$APO = SAPO(LCPDAT208),$JERK = SJERK(LCPDAT208),$COLLMON_TOL_PRO[1] = USE_CM_PRO_VALUES(0)
;ENDFOLD

;FOLD SLIN P209 Vel=2 m/s CPDAT209 Tool[4]:Microflown3D Base[2]:straight_sol;%{PE}
;FOLD Parameters ;%{h}
;Params IlfProvider=kukaroboter.basistech.inlineforms.movement.spline; Kuka.IsGlobalPoint=False; Kuka.PointName=P209; Kuka.BlendingEnabled=False; Kuka.MoveDataName=CPDAT209; Kuka.VelocityPath=2.000; Kuka.VelocityFieldEnabled=True; Kuka.ColDetectFieldEnabled=True; Kuka.CurrentCDSetIndex=0; Kuka.MovementParameterFieldEnabled=True; IlfCommand=SLIN
;ENDFOLD
SLIN XP209 WITH $VEL = SVEL_CP(2.0, , LCPDAT209),$TOOL = STOOL2(FP209),$BASE = SBASE(FP209.BASE_NO),$IPO_MODE = SIPO_MODE(FP209.IPO_FRAME),$LOAD = SLOAD(FP209.TOOL_NO),$ACC = SACC_CP(LCPDAT209),$ORI_TYPE = SORI_TYP(LCPDAT209),$APO = SAPO(LCPDAT209),$JERK = SJERK(LCPDAT209),$COLLMON_TOL_PRO[1] = USE_CM_PRO_VALUES(0)
;ENDFOLD

;FOLD SLIN P210 Vel=2 m/s CPDAT210 Tool[4]:Microflown3D Base[2]:straight_sol;%{PE}
;FOLD Parameters ;%{h}
;Params IlfProvider=kukaroboter.basistech.inlineforms.movement.spline; Kuka.IsGlobalPoint=False; Kuka.PointName=P210; Kuka.BlendingEnabled=False; Kuka.MoveDataName=CPDAT210; Kuka.VelocityPath=2.000; Kuka.VelocityFieldEnabled=True; Kuka.ColDetectFieldEnabled=True; Kuka.CurrentCDSetIndex=0; Kuka.MovementParameterFieldEnabled=True; IlfCommand=SLIN
;ENDFOLD
SLIN XP210 WITH $VEL = SVEL_CP(2.0, , LCPDAT210),$TOOL = STOOL2(FP210),$BASE = SBASE(FP210.BASE_NO),$IPO_MODE = SIPO_MODE(FP210.IPO_FRAME),$LOAD = SLOAD(FP210.TOOL_NO),$ACC = SACC_CP(LCPDAT210),$ORI_TYPE = SORI_TYP(LCPDAT210),$APO = SAPO(LCPDAT210),$JERK = SJERK(LCPDAT210),$COLLMON_TOL_PRO[1] = USE_CM_PRO_VALUES(0)
;ENDFOLD

;FOLD SLIN P211 Vel=2 m/s CPDAT211 Tool[4]:Microflown3D Base[2]:straight_sol;%{PE}
;FOLD Parameters ;%{h}
;Params IlfProvider=kukaroboter.basistech.inlineforms.movement.spline; Kuka.IsGlobalPoint=False; Kuka.PointName=P211; Kuka.BlendingEnabled=False; Kuka.MoveDataName=CPDAT211; Kuka.VelocityPath=2.000; Kuka.VelocityFieldEnabled=True; Kuka.ColDetectFieldEnabled=True; Kuka.CurrentCDSetIndex=0; Kuka.MovementParameterFieldEnabled=True; IlfCommand=SLIN
;ENDFOLD
SLIN XP211 WITH $VEL = SVEL_CP(2.0, , LCPDAT211),$TOOL = STOOL2(FP211),$BASE = SBASE(FP211.BASE_NO),$IPO_MODE = SIPO_MODE(FP211.IPO_FRAME),$LOAD = SLOAD(FP211.TOOL_NO),$ACC = SACC_CP(LCPDAT211),$ORI_TYPE = SORI_TYP(LCPDAT211),$APO = SAPO(LCPDAT211),$JERK = SJERK(LCPDAT211),$COLLMON_TOL_PRO[1] = USE_CM_PRO_VALUES(0)
;ENDFOLD

;FOLD SLIN P212 Vel=2 m/s CPDAT212 Tool[4]:Microflown3D Base[2]:straight_sol;%{PE}
;FOLD Parameters ;%{h}
;Params IlfProvider=kukaroboter.basistech.inlineforms.movement.spline; Kuka.IsGlobalPoint=False; Kuka.PointName=P212; Kuka.BlendingEnabled=False; Kuka.MoveDataName=CPDAT212; Kuka.VelocityPath=2.000; Kuka.VelocityFieldEnabled=True; Kuka.ColDetectFieldEnabled=True; Kuka.CurrentCDSetIndex=0; Kuka.MovementParameterFieldEnabled=True; IlfCommand=SLIN
;ENDFOLD
SLIN XP212 WITH $VEL = SVEL_CP(2.0, , LCPDAT212),$TOOL = STOOL2(FP212),$BASE = SBASE(FP212.BASE_NO),$IPO_MODE = SIPO_MODE(FP212.IPO_FRAME),$LOAD = SLOAD(FP212.TOOL_NO),$ACC = SACC_CP(LCPDAT212),$ORI_TYPE = SORI_TYP(LCPDAT212),$APO = SAPO(LCPDAT212),$JERK = SJERK(LCPDAT212),$COLLMON_TOL_PRO[1] = USE_CM_PRO_VALUES(0)
;ENDFOLD

;FOLD SLIN P213 Vel=2 m/s CPDAT213 Tool[4]:Microflown3D Base[2]:straight_sol;%{PE}
;FOLD Parameters ;%{h}
;Params IlfProvider=kukaroboter.basistech.inlineforms.movement.spline; Kuka.IsGlobalPoint=False; Kuka.PointName=P213; Kuka.BlendingEnabled=False; Kuka.MoveDataName=CPDAT213; Kuka.VelocityPath=2.000; Kuka.VelocityFieldEnabled=True; Kuka.ColDetectFieldEnabled=True; Kuka.CurrentCDSetIndex=0; Kuka.MovementParameterFieldEnabled=True; IlfCommand=SLIN
;ENDFOLD
SLIN XP213 WITH $VEL = SVEL_CP(2.0, , LCPDAT213),$TOOL = STOOL2(FP213),$BASE = SBASE(FP213.BASE_NO),$IPO_MODE = SIPO_MODE(FP213.IPO_FRAME),$LOAD = SLOAD(FP213.TOOL_NO),$ACC = SACC_CP(LCPDAT213),$ORI_TYPE = SORI_TYP(LCPDAT213),$APO = SAPO(LCPDAT213),$JERK = SJERK(LCPDAT213),$COLLMON_TOL_PRO[1] = USE_CM_PRO_VALUES(0)
;ENDFOLD

;FOLD SLIN P214 Vel=2 m/s CPDAT214 Tool[4]:Microflown3D Base[2]:straight_sol;%{PE}
;FOLD Parameters ;%{h}
;Params IlfProvider=kukaroboter.basistech.inlineforms.movement.spline; Kuka.IsGlobalPoint=False; Kuka.PointName=P214; Kuka.BlendingEnabled=False; Kuka.MoveDataName=CPDAT214; Kuka.VelocityPath=2.000; Kuka.VelocityFieldEnabled=True; Kuka.ColDetectFieldEnabled=True; Kuka.CurrentCDSetIndex=0; Kuka.MovementParameterFieldEnabled=True; IlfCommand=SLIN
;ENDFOLD
SLIN XP214 WITH $VEL = SVEL_CP(2.0, , LCPDAT214),$TOOL = STOOL2(FP214),$BASE = SBASE(FP214.BASE_NO),$IPO_MODE = SIPO_MODE(FP214.IPO_FRAME),$LOAD = SLOAD(FP214.TOOL_NO),$ACC = SACC_CP(LCPDAT214),$ORI_TYPE = SORI_TYP(LCPDAT214),$APO = SAPO(LCPDAT214),$JERK = SJERK(LCPDAT214),$COLLMON_TOL_PRO[1] = USE_CM_PRO_VALUES(0)
;ENDFOLD

;FOLD SLIN P215 Vel=2 m/s CPDAT215 Tool[4]:Microflown3D Base[2]:straight_sol;%{PE}
;FOLD Parameters ;%{h}
;Params IlfProvider=kukaroboter.basistech.inlineforms.movement.spline; Kuka.IsGlobalPoint=False; Kuka.PointName=P215; Kuka.BlendingEnabled=False; Kuka.MoveDataName=CPDAT215; Kuka.VelocityPath=2.000; Kuka.VelocityFieldEnabled=True; Kuka.ColDetectFieldEnabled=True; Kuka.CurrentCDSetIndex=0; Kuka.MovementParameterFieldEnabled=True; IlfCommand=SLIN
;ENDFOLD
SLIN XP215 WITH $VEL = SVEL_CP(2.0, , LCPDAT215),$TOOL = STOOL2(FP215),$BASE = SBASE(FP215.BASE_NO),$IPO_MODE = SIPO_MODE(FP215.IPO_FRAME),$LOAD = SLOAD(FP215.TOOL_NO),$ACC = SACC_CP(LCPDAT215),$ORI_TYPE = SORI_TYP(LCPDAT215),$APO = SAPO(LCPDAT215),$JERK = SJERK(LCPDAT215),$COLLMON_TOL_PRO[1] = USE_CM_PRO_VALUES(0)
;ENDFOLD

;FOLD SLIN P216 Vel=2 m/s CPDAT216 Tool[4]:Microflown3D Base[2]:straight_sol;%{PE}
;FOLD Parameters ;%{h}
;Params IlfProvider=kukaroboter.basistech.inlineforms.movement.spline; Kuka.IsGlobalPoint=False; Kuka.PointName=P216; Kuka.BlendingEnabled=False; Kuka.MoveDataName=CPDAT216; Kuka.VelocityPath=2.000; Kuka.VelocityFieldEnabled=True; Kuka.ColDetectFieldEnabled=True; Kuka.CurrentCDSetIndex=0; Kuka.MovementParameterFieldEnabled=True; IlfCommand=SLIN
;ENDFOLD
SLIN XP216 WITH $VEL = SVEL_CP(2.0, , LCPDAT216),$TOOL = STOOL2(FP216),$BASE = SBASE(FP216.BASE_NO),$IPO_MODE = SIPO_MODE(FP216.IPO_FRAME),$LOAD = SLOAD(FP216.TOOL_NO),$ACC = SACC_CP(LCPDAT216),$ORI_TYPE = SORI_TYP(LCPDAT216),$APO = SAPO(LCPDAT216),$JERK = SJERK(LCPDAT216),$COLLMON_TOL_PRO[1] = USE_CM_PRO_VALUES(0)
;ENDFOLD

;FOLD SLIN P217 Vel=2 m/s CPDAT217 Tool[4]:Microflown3D Base[2]:straight_sol;%{PE}
;FOLD Parameters ;%{h}
;Params IlfProvider=kukaroboter.basistech.inlineforms.movement.spline; Kuka.IsGlobalPoint=False; Kuka.PointName=P217; Kuka.BlendingEnabled=False; Kuka.MoveDataName=CPDAT217; Kuka.VelocityPath=2.000; Kuka.VelocityFieldEnabled=True; Kuka.ColDetectFieldEnabled=True; Kuka.CurrentCDSetIndex=0; Kuka.MovementParameterFieldEnabled=True; IlfCommand=SLIN
;ENDFOLD
SLIN XP217 WITH $VEL = SVEL_CP(2.0, , LCPDAT217),$TOOL = STOOL2(FP217),$BASE = SBASE(FP217.BASE_NO),$IPO_MODE = SIPO_MODE(FP217.IPO_FRAME),$LOAD = SLOAD(FP217.TOOL_NO),$ACC = SACC_CP(LCPDAT217),$ORI_TYPE = SORI_TYP(LCPDAT217),$APO = SAPO(LCPDAT217),$JERK = SJERK(LCPDAT217),$COLLMON_TOL_PRO[1] = USE_CM_PRO_VALUES(0)
;ENDFOLD

;FOLD SLIN P218 Vel=2 m/s CPDAT218 Tool[4]:Microflown3D Base[2]:straight_sol;%{PE}
;FOLD Parameters ;%{h}
;Params IlfProvider=kukaroboter.basistech.inlineforms.movement.spline; Kuka.IsGlobalPoint=False; Kuka.PointName=P218; Kuka.BlendingEnabled=False; Kuka.MoveDataName=CPDAT218; Kuka.VelocityPath=2.000; Kuka.VelocityFieldEnabled=True; Kuka.ColDetectFieldEnabled=True; Kuka.CurrentCDSetIndex=0; Kuka.MovementParameterFieldEnabled=True; IlfCommand=SLIN
;ENDFOLD
SLIN XP218 WITH $VEL = SVEL_CP(2.0, , LCPDAT218),$TOOL = STOOL2(FP218),$BASE = SBASE(FP218.BASE_NO),$IPO_MODE = SIPO_MODE(FP218.IPO_FRAME),$LOAD = SLOAD(FP218.TOOL_NO),$ACC = SACC_CP(LCPDAT218),$ORI_TYPE = SORI_TYP(LCPDAT218),$APO = SAPO(LCPDAT218),$JERK = SJERK(LCPDAT218),$COLLMON_TOL_PRO[1] = USE_CM_PRO_VALUES(0)
;ENDFOLD

;FOLD SLIN P219 Vel=2 m/s CPDAT219 Tool[4]:Microflown3D Base[2]:straight_sol;%{PE}
;FOLD Parameters ;%{h}
;Params IlfProvider=kukaroboter.basistech.inlineforms.movement.spline; Kuka.IsGlobalPoint=False; Kuka.PointName=P219; Kuka.BlendingEnabled=False; Kuka.MoveDataName=CPDAT219; Kuka.VelocityPath=2.000; Kuka.VelocityFieldEnabled=True; Kuka.ColDetectFieldEnabled=True; Kuka.CurrentCDSetIndex=0; Kuka.MovementParameterFieldEnabled=True; IlfCommand=SLIN
;ENDFOLD
SLIN XP219 WITH $VEL = SVEL_CP(2.0, , LCPDAT219),$TOOL = STOOL2(FP219),$BASE = SBASE(FP219.BASE_NO),$IPO_MODE = SIPO_MODE(FP219.IPO_FRAME),$LOAD = SLOAD(FP219.TOOL_NO),$ACC = SACC_CP(LCPDAT219),$ORI_TYPE = SORI_TYP(LCPDAT219),$APO = SAPO(LCPDAT219),$JERK = SJERK(LCPDAT219),$COLLMON_TOL_PRO[1] = USE_CM_PRO_VALUES(0)
;ENDFOLD

;FOLD SLIN P220 Vel=2 m/s CPDAT220 Tool[4]:Microflown3D Base[2]:straight_sol;%{PE}
;FOLD Parameters ;%{h}
;Params IlfProvider=kukaroboter.basistech.inlineforms.movement.spline; Kuka.IsGlobalPoint=False; Kuka.PointName=P220; Kuka.BlendingEnabled=False; Kuka.MoveDataName=CPDAT220; Kuka.VelocityPath=2.000; Kuka.VelocityFieldEnabled=True; Kuka.ColDetectFieldEnabled=True; Kuka.CurrentCDSetIndex=0; Kuka.MovementParameterFieldEnabled=True; IlfCommand=SLIN
;ENDFOLD
SLIN XP220 WITH $VEL = SVEL_CP(2.0, , LCPDAT220),$TOOL = STOOL2(FP220),$BASE = SBASE(FP220.BASE_NO),$IPO_MODE = SIPO_MODE(FP220.IPO_FRAME),$LOAD = SLOAD(FP220.TOOL_NO),$ACC = SACC_CP(LCPDAT220),$ORI_TYPE = SORI_TYP(LCPDAT220),$APO = SAPO(LCPDAT220),$JERK = SJERK(LCPDAT220),$COLLMON_TOL_PRO[1] = USE_CM_PRO_VALUES(0)
;ENDFOLD

;FOLD SLIN P221 Vel=2 m/s CPDAT221 Tool[4]:Microflown3D Base[2]:straight_sol;%{PE}
;FOLD Parameters ;%{h}
;Params IlfProvider=kukaroboter.basistech.inlineforms.movement.spline; Kuka.IsGlobalPoint=False; Kuka.PointName=P221; Kuka.BlendingEnabled=False; Kuka.MoveDataName=CPDAT221; Kuka.VelocityPath=2.000; Kuka.VelocityFieldEnabled=True; Kuka.ColDetectFieldEnabled=True; Kuka.CurrentCDSetIndex=0; Kuka.MovementParameterFieldEnabled=True; IlfCommand=SLIN
;ENDFOLD
SLIN XP221 WITH $VEL = SVEL_CP(2.0, , LCPDAT221),$TOOL = STOOL2(FP221),$BASE = SBASE(FP221.BASE_NO),$IPO_MODE = SIPO_MODE(FP221.IPO_FRAME),$LOAD = SLOAD(FP221.TOOL_NO),$ACC = SACC_CP(LCPDAT221),$ORI_TYPE = SORI_TYP(LCPDAT221),$APO = SAPO(LCPDAT221),$JERK = SJERK(LCPDAT221),$COLLMON_TOL_PRO[1] = USE_CM_PRO_VALUES(0)
;ENDFOLD

;FOLD SLIN P222 Vel=2 m/s CPDAT222 Tool[4]:Microflown3D Base[2]:straight_sol;%{PE}
;FOLD Parameters ;%{h}
;Params IlfProvider=kukaroboter.basistech.inlineforms.movement.spline; Kuka.IsGlobalPoint=False; Kuka.PointName=P222; Kuka.BlendingEnabled=False; Kuka.MoveDataName=CPDAT222; Kuka.VelocityPath=2.000; Kuka.VelocityFieldEnabled=True; Kuka.ColDetectFieldEnabled=True; Kuka.CurrentCDSetIndex=0; Kuka.MovementParameterFieldEnabled=True; IlfCommand=SLIN
;ENDFOLD
SLIN XP222 WITH $VEL = SVEL_CP(2.0, , LCPDAT222),$TOOL = STOOL2(FP222),$BASE = SBASE(FP222.BASE_NO),$IPO_MODE = SIPO_MODE(FP222.IPO_FRAME),$LOAD = SLOAD(FP222.TOOL_NO),$ACC = SACC_CP(LCPDAT222),$ORI_TYPE = SORI_TYP(LCPDAT222),$APO = SAPO(LCPDAT222),$JERK = SJERK(LCPDAT222),$COLLMON_TOL_PRO[1] = USE_CM_PRO_VALUES(0)
;ENDFOLD

;FOLD SLIN P223 Vel=2 m/s CPDAT223 Tool[4]:Microflown3D Base[2]:straight_sol;%{PE}
;FOLD Parameters ;%{h}
;Params IlfProvider=kukaroboter.basistech.inlineforms.movement.spline; Kuka.IsGlobalPoint=False; Kuka.PointName=P223; Kuka.BlendingEnabled=False; Kuka.MoveDataName=CPDAT223; Kuka.VelocityPath=2.000; Kuka.VelocityFieldEnabled=True; Kuka.ColDetectFieldEnabled=True; Kuka.CurrentCDSetIndex=0; Kuka.MovementParameterFieldEnabled=True; IlfCommand=SLIN
;ENDFOLD
SLIN XP223 WITH $VEL = SVEL_CP(2.0, , LCPDAT223),$TOOL = STOOL2(FP223),$BASE = SBASE(FP223.BASE_NO),$IPO_MODE = SIPO_MODE(FP223.IPO_FRAME),$LOAD = SLOAD(FP223.TOOL_NO),$ACC = SACC_CP(LCPDAT223),$ORI_TYPE = SORI_TYP(LCPDAT223),$APO = SAPO(LCPDAT223),$JERK = SJERK(LCPDAT223),$COLLMON_TOL_PRO[1] = USE_CM_PRO_VALUES(0)
;ENDFOLD

;FOLD SLIN P224 Vel=2 m/s CPDAT224 Tool[4]:Microflown3D Base[2]:straight_sol;%{PE}
;FOLD Parameters ;%{h}
;Params IlfProvider=kukaroboter.basistech.inlineforms.movement.spline; Kuka.IsGlobalPoint=False; Kuka.PointName=P224; Kuka.BlendingEnabled=False; Kuka.MoveDataName=CPDAT224; Kuka.VelocityPath=2.000; Kuka.VelocityFieldEnabled=True; Kuka.ColDetectFieldEnabled=True; Kuka.CurrentCDSetIndex=0; Kuka.MovementParameterFieldEnabled=True; IlfCommand=SLIN
;ENDFOLD
SLIN XP224 WITH $VEL = SVEL_CP(2.0, , LCPDAT224),$TOOL = STOOL2(FP224),$BASE = SBASE(FP224.BASE_NO),$IPO_MODE = SIPO_MODE(FP224.IPO_FRAME),$LOAD = SLOAD(FP224.TOOL_NO),$ACC = SACC_CP(LCPDAT224),$ORI_TYPE = SORI_TYP(LCPDAT224),$APO = SAPO(LCPDAT224),$JERK = SJERK(LCPDAT224),$COLLMON_TOL_PRO[1] = USE_CM_PRO_VALUES(0)
;ENDFOLD

;FOLD SLIN P225 Vel=2 m/s CPDAT225 Tool[4]:Microflown3D Base[2]:straight_sol;%{PE}
;FOLD Parameters ;%{h}
;Params IlfProvider=kukaroboter.basistech.inlineforms.movement.spline; Kuka.IsGlobalPoint=False; Kuka.PointName=P225; Kuka.BlendingEnabled=False; Kuka.MoveDataName=CPDAT225; Kuka.VelocityPath=2.000; Kuka.VelocityFieldEnabled=True; Kuka.ColDetectFieldEnabled=True; Kuka.CurrentCDSetIndex=0; Kuka.MovementParameterFieldEnabled=True; IlfCommand=SLIN
;ENDFOLD
SLIN XP225 WITH $VEL = SVEL_CP(2.0, , LCPDAT225),$TOOL = STOOL2(FP225),$BASE = SBASE(FP225.BASE_NO),$IPO_MODE = SIPO_MODE(FP225.IPO_FRAME),$LOAD = SLOAD(FP225.TOOL_NO),$ACC = SACC_CP(LCPDAT225),$ORI_TYPE = SORI_TYP(LCPDAT225),$APO = SAPO(LCPDAT225),$JERK = SJERK(LCPDAT225),$COLLMON_TOL_PRO[1] = USE_CM_PRO_VALUES(0)
;ENDFOLD

;FOLD SLIN P226 Vel=2 m/s CPDAT226 Tool[4]:Microflown3D Base[2]:straight_sol;%{PE}
;FOLD Parameters ;%{h}
;Params IlfProvider=kukaroboter.basistech.inlineforms.movement.spline; Kuka.IsGlobalPoint=False; Kuka.PointName=P226; Kuka.BlendingEnabled=False; Kuka.MoveDataName=CPDAT226; Kuka.VelocityPath=2.000; Kuka.VelocityFieldEnabled=True; Kuka.ColDetectFieldEnabled=True; Kuka.CurrentCDSetIndex=0; Kuka.MovementParameterFieldEnabled=True; IlfCommand=SLIN
;ENDFOLD
SLIN XP226 WITH $VEL = SVEL_CP(2.0, , LCPDAT226),$TOOL = STOOL2(FP226),$BASE = SBASE(FP226.BASE_NO),$IPO_MODE = SIPO_MODE(FP226.IPO_FRAME),$LOAD = SLOAD(FP226.TOOL_NO),$ACC = SACC_CP(LCPDAT226),$ORI_TYPE = SORI_TYP(LCPDAT226),$APO = SAPO(LCPDAT226),$JERK = SJERK(LCPDAT226),$COLLMON_TOL_PRO[1] = USE_CM_PRO_VALUES(0)
;ENDFOLD

;FOLD SLIN P227 Vel=2 m/s CPDAT227 Tool[4]:Microflown3D Base[2]:straight_sol;%{PE}
;FOLD Parameters ;%{h}
;Params IlfProvider=kukaroboter.basistech.inlineforms.movement.spline; Kuka.IsGlobalPoint=False; Kuka.PointName=P227; Kuka.BlendingEnabled=False; Kuka.MoveDataName=CPDAT227; Kuka.VelocityPath=2.000; Kuka.VelocityFieldEnabled=True; Kuka.ColDetectFieldEnabled=True; Kuka.CurrentCDSetIndex=0; Kuka.MovementParameterFieldEnabled=True; IlfCommand=SLIN
;ENDFOLD
SLIN XP227 WITH $VEL = SVEL_CP(2.0, , LCPDAT227),$TOOL = STOOL2(FP227),$BASE = SBASE(FP227.BASE_NO),$IPO_MODE = SIPO_MODE(FP227.IPO_FRAME),$LOAD = SLOAD(FP227.TOOL_NO),$ACC = SACC_CP(LCPDAT227),$ORI_TYPE = SORI_TYP(LCPDAT227),$APO = SAPO(LCPDAT227),$JERK = SJERK(LCPDAT227),$COLLMON_TOL_PRO[1] = USE_CM_PRO_VALUES(0)
;ENDFOLD

;FOLD SLIN P228 Vel=2 m/s CPDAT228 Tool[4]:Microflown3D Base[2]:straight_sol;%{PE}
;FOLD Parameters ;%{h}
;Params IlfProvider=kukaroboter.basistech.inlineforms.movement.spline; Kuka.IsGlobalPoint=False; Kuka.PointName=P228; Kuka.BlendingEnabled=False; Kuka.MoveDataName=CPDAT228; Kuka.VelocityPath=2.000; Kuka.VelocityFieldEnabled=True; Kuka.ColDetectFieldEnabled=True; Kuka.CurrentCDSetIndex=0; Kuka.MovementParameterFieldEnabled=True; IlfCommand=SLIN
;ENDFOLD
SLIN XP228 WITH $VEL = SVEL_CP(2.0, , LCPDAT228),$TOOL = STOOL2(FP228),$BASE = SBASE(FP228.BASE_NO),$IPO_MODE = SIPO_MODE(FP228.IPO_FRAME),$LOAD = SLOAD(FP228.TOOL_NO),$ACC = SACC_CP(LCPDAT228),$ORI_TYPE = SORI_TYP(LCPDAT228),$APO = SAPO(LCPDAT228),$JERK = SJERK(LCPDAT228),$COLLMON_TOL_PRO[1] = USE_CM_PRO_VALUES(0)
;ENDFOLD

;FOLD SLIN P229 Vel=2 m/s CPDAT229 Tool[4]:Microflown3D Base[2]:straight_sol;%{PE}
;FOLD Parameters ;%{h}
;Params IlfProvider=kukaroboter.basistech.inlineforms.movement.spline; Kuka.IsGlobalPoint=False; Kuka.PointName=P229; Kuka.BlendingEnabled=False; Kuka.MoveDataName=CPDAT229; Kuka.VelocityPath=2.000; Kuka.VelocityFieldEnabled=True; Kuka.ColDetectFieldEnabled=True; Kuka.CurrentCDSetIndex=0; Kuka.MovementParameterFieldEnabled=True; IlfCommand=SLIN
;ENDFOLD
SLIN XP229 WITH $VEL = SVEL_CP(2.0, , LCPDAT229),$TOOL = STOOL2(FP229),$BASE = SBASE(FP229.BASE_NO),$IPO_MODE = SIPO_MODE(FP229.IPO_FRAME),$LOAD = SLOAD(FP229.TOOL_NO),$ACC = SACC_CP(LCPDAT229),$ORI_TYPE = SORI_TYP(LCPDAT229),$APO = SAPO(LCPDAT229),$JERK = SJERK(LCPDAT229),$COLLMON_TOL_PRO[1] = USE_CM_PRO_VALUES(0)
;ENDFOLD

;FOLD SLIN P230 Vel=2 m/s CPDAT230 Tool[4]:Microflown3D Base[2]:straight_sol;%{PE}
;FOLD Parameters ;%{h}
;Params IlfProvider=kukaroboter.basistech.inlineforms.movement.spline; Kuka.IsGlobalPoint=False; Kuka.PointName=P230; Kuka.BlendingEnabled=False; Kuka.MoveDataName=CPDAT230; Kuka.VelocityPath=2.000; Kuka.VelocityFieldEnabled=True; Kuka.ColDetectFieldEnabled=True; Kuka.CurrentCDSetIndex=0; Kuka.MovementParameterFieldEnabled=True; IlfCommand=SLIN
;ENDFOLD
SLIN XP230 WITH $VEL = SVEL_CP(2.0, , LCPDAT230),$TOOL = STOOL2(FP230),$BASE = SBASE(FP230.BASE_NO),$IPO_MODE = SIPO_MODE(FP230.IPO_FRAME),$LOAD = SLOAD(FP230.TOOL_NO),$ACC = SACC_CP(LCPDAT230),$ORI_TYPE = SORI_TYP(LCPDAT230),$APO = SAPO(LCPDAT230),$JERK = SJERK(LCPDAT230),$COLLMON_TOL_PRO[1] = USE_CM_PRO_VALUES(0)
;ENDFOLD

;FOLD SLIN P231 Vel=2 m/s CPDAT231 Tool[4]:Microflown3D Base[2]:straight_sol;%{PE}
;FOLD Parameters ;%{h}
;Params IlfProvider=kukaroboter.basistech.inlineforms.movement.spline; Kuka.IsGlobalPoint=False; Kuka.PointName=P231; Kuka.BlendingEnabled=False; Kuka.MoveDataName=CPDAT231; Kuka.VelocityPath=2.000; Kuka.VelocityFieldEnabled=True; Kuka.ColDetectFieldEnabled=True; Kuka.CurrentCDSetIndex=0; Kuka.MovementParameterFieldEnabled=True; IlfCommand=SLIN
;ENDFOLD
SLIN XP231 WITH $VEL = SVEL_CP(2.0, , LCPDAT231),$TOOL = STOOL2(FP231),$BASE = SBASE(FP231.BASE_NO),$IPO_MODE = SIPO_MODE(FP231.IPO_FRAME),$LOAD = SLOAD(FP231.TOOL_NO),$ACC = SACC_CP(LCPDAT231),$ORI_TYPE = SORI_TYP(LCPDAT231),$APO = SAPO(LCPDAT231),$JERK = SJERK(LCPDAT231),$COLLMON_TOL_PRO[1] = USE_CM_PRO_VALUES(0)
;ENDFOLD

;FOLD SLIN P232 Vel=2 m/s CPDAT232 Tool[4]:Microflown3D Base[2]:straight_sol;%{PE}
;FOLD Parameters ;%{h}
;Params IlfProvider=kukaroboter.basistech.inlineforms.movement.spline; Kuka.IsGlobalPoint=False; Kuka.PointName=P232; Kuka.BlendingEnabled=False; Kuka.MoveDataName=CPDAT232; Kuka.VelocityPath=2.000; Kuka.VelocityFieldEnabled=True; Kuka.ColDetectFieldEnabled=True; Kuka.CurrentCDSetIndex=0; Kuka.MovementParameterFieldEnabled=True; IlfCommand=SLIN
;ENDFOLD
SLIN XP232 WITH $VEL = SVEL_CP(2.0, , LCPDAT232),$TOOL = STOOL2(FP232),$BASE = SBASE(FP232.BASE_NO),$IPO_MODE = SIPO_MODE(FP232.IPO_FRAME),$LOAD = SLOAD(FP232.TOOL_NO),$ACC = SACC_CP(LCPDAT232),$ORI_TYPE = SORI_TYP(LCPDAT232),$APO = SAPO(LCPDAT232),$JERK = SJERK(LCPDAT232),$COLLMON_TOL_PRO[1] = USE_CM_PRO_VALUES(0)
;ENDFOLD

;FOLD SLIN P233 Vel=2 m/s CPDAT233 Tool[4]:Microflown3D Base[2]:straight_sol;%{PE}
;FOLD Parameters ;%{h}
;Params IlfProvider=kukaroboter.basistech.inlineforms.movement.spline; Kuka.IsGlobalPoint=False; Kuka.PointName=P233; Kuka.BlendingEnabled=False; Kuka.MoveDataName=CPDAT233; Kuka.VelocityPath=2.000; Kuka.VelocityFieldEnabled=True; Kuka.ColDetectFieldEnabled=True; Kuka.CurrentCDSetIndex=0; Kuka.MovementParameterFieldEnabled=True; IlfCommand=SLIN
;ENDFOLD
SLIN XP233 WITH $VEL = SVEL_CP(2.0, , LCPDAT233),$TOOL = STOOL2(FP233),$BASE = SBASE(FP233.BASE_NO),$IPO_MODE = SIPO_MODE(FP233.IPO_FRAME),$LOAD = SLOAD(FP233.TOOL_NO),$ACC = SACC_CP(LCPDAT233),$ORI_TYPE = SORI_TYP(LCPDAT233),$APO = SAPO(LCPDAT233),$JERK = SJERK(LCPDAT233),$COLLMON_TOL_PRO[1] = USE_CM_PRO_VALUES(0)
;ENDFOLD

;FOLD SLIN P234 Vel=2 m/s CPDAT234 Tool[4]:Microflown3D Base[2]:straight_sol;%{PE}
;FOLD Parameters ;%{h}
;Params IlfProvider=kukaroboter.basistech.inlineforms.movement.spline; Kuka.IsGlobalPoint=False; Kuka.PointName=P234; Kuka.BlendingEnabled=False; Kuka.MoveDataName=CPDAT234; Kuka.VelocityPath=2.000; Kuka.VelocityFieldEnabled=True; Kuka.ColDetectFieldEnabled=True; Kuka.CurrentCDSetIndex=0; Kuka.MovementParameterFieldEnabled=True; IlfCommand=SLIN
;ENDFOLD
SLIN XP234 WITH $VEL = SVEL_CP(2.0, , LCPDAT234),$TOOL = STOOL2(FP234),$BASE = SBASE(FP234.BASE_NO),$IPO_MODE = SIPO_MODE(FP234.IPO_FRAME),$LOAD = SLOAD(FP234.TOOL_NO),$ACC = SACC_CP(LCPDAT234),$ORI_TYPE = SORI_TYP(LCPDAT234),$APO = SAPO(LCPDAT234),$JERK = SJERK(LCPDAT234),$COLLMON_TOL_PRO[1] = USE_CM_PRO_VALUES(0)
;ENDFOLD

;FOLD SLIN P235 Vel=2 m/s CPDAT235 Tool[4]:Microflown3D Base[2]:straight_sol;%{PE}
;FOLD Parameters ;%{h}
;Params IlfProvider=kukaroboter.basistech.inlineforms.movement.spline; Kuka.IsGlobalPoint=False; Kuka.PointName=P235; Kuka.BlendingEnabled=False; Kuka.MoveDataName=CPDAT235; Kuka.VelocityPath=2.000; Kuka.VelocityFieldEnabled=True; Kuka.ColDetectFieldEnabled=True; Kuka.CurrentCDSetIndex=0; Kuka.MovementParameterFieldEnabled=True; IlfCommand=SLIN
;ENDFOLD
SLIN XP235 WITH $VEL = SVEL_CP(2.0, , LCPDAT235),$TOOL = STOOL2(FP235),$BASE = SBASE(FP235.BASE_NO),$IPO_MODE = SIPO_MODE(FP235.IPO_FRAME),$LOAD = SLOAD(FP235.TOOL_NO),$ACC = SACC_CP(LCPDAT235),$ORI_TYPE = SORI_TYP(LCPDAT235),$APO = SAPO(LCPDAT235),$JERK = SJERK(LCPDAT235),$COLLMON_TOL_PRO[1] = USE_CM_PRO_VALUES(0)
;ENDFOLD

;FOLD SLIN P236 Vel=2 m/s CPDAT236 Tool[4]:Microflown3D Base[2]:straight_sol;%{PE}
;FOLD Parameters ;%{h}
;Params IlfProvider=kukaroboter.basistech.inlineforms.movement.spline; Kuka.IsGlobalPoint=False; Kuka.PointName=P236; Kuka.BlendingEnabled=False; Kuka.MoveDataName=CPDAT236; Kuka.VelocityPath=2.000; Kuka.VelocityFieldEnabled=True; Kuka.ColDetectFieldEnabled=True; Kuka.CurrentCDSetIndex=0; Kuka.MovementParameterFieldEnabled=True; IlfCommand=SLIN
;ENDFOLD
SLIN XP236 WITH $VEL = SVEL_CP(2.0, , LCPDAT236),$TOOL = STOOL2(FP236),$BASE = SBASE(FP236.BASE_NO),$IPO_MODE = SIPO_MODE(FP236.IPO_FRAME),$LOAD = SLOAD(FP236.TOOL_NO),$ACC = SACC_CP(LCPDAT236),$ORI_TYPE = SORI_TYP(LCPDAT236),$APO = SAPO(LCPDAT236),$JERK = SJERK(LCPDAT236),$COLLMON_TOL_PRO[1] = USE_CM_PRO_VALUES(0)
;ENDFOLD

;FOLD SLIN P237 Vel=2 m/s CPDAT237 Tool[4]:Microflown3D Base[2]:straight_sol;%{PE}
;FOLD Parameters ;%{h}
;Params IlfProvider=kukaroboter.basistech.inlineforms.movement.spline; Kuka.IsGlobalPoint=False; Kuka.PointName=P237; Kuka.BlendingEnabled=False; Kuka.MoveDataName=CPDAT237; Kuka.VelocityPath=2.000; Kuka.VelocityFieldEnabled=True; Kuka.ColDetectFieldEnabled=True; Kuka.CurrentCDSetIndex=0; Kuka.MovementParameterFieldEnabled=True; IlfCommand=SLIN
;ENDFOLD
SLIN XP237 WITH $VEL = SVEL_CP(2.0, , LCPDAT237),$TOOL = STOOL2(FP237),$BASE = SBASE(FP237.BASE_NO),$IPO_MODE = SIPO_MODE(FP237.IPO_FRAME),$LOAD = SLOAD(FP237.TOOL_NO),$ACC = SACC_CP(LCPDAT237),$ORI_TYPE = SORI_TYP(LCPDAT237),$APO = SAPO(LCPDAT237),$JERK = SJERK(LCPDAT237),$COLLMON_TOL_PRO[1] = USE_CM_PRO_VALUES(0)
;ENDFOLD

;FOLD SLIN P238 Vel=2 m/s CPDAT238 Tool[4]:Microflown3D Base[2]:straight_sol;%{PE}
;FOLD Parameters ;%{h}
;Params IlfProvider=kukaroboter.basistech.inlineforms.movement.spline; Kuka.IsGlobalPoint=False; Kuka.PointName=P238; Kuka.BlendingEnabled=False; Kuka.MoveDataName=CPDAT238; Kuka.VelocityPath=2.000; Kuka.VelocityFieldEnabled=True; Kuka.ColDetectFieldEnabled=True; Kuka.CurrentCDSetIndex=0; Kuka.MovementParameterFieldEnabled=True; IlfCommand=SLIN
;ENDFOLD
SLIN XP238 WITH $VEL = SVEL_CP(2.0, , LCPDAT238),$TOOL = STOOL2(FP238),$BASE = SBASE(FP238.BASE_NO),$IPO_MODE = SIPO_MODE(FP238.IPO_FRAME),$LOAD = SLOAD(FP238.TOOL_NO),$ACC = SACC_CP(LCPDAT238),$ORI_TYPE = SORI_TYP(LCPDAT238),$APO = SAPO(LCPDAT238),$JERK = SJERK(LCPDAT238),$COLLMON_TOL_PRO[1] = USE_CM_PRO_VALUES(0)
;ENDFOLD

;FOLD SLIN P239 Vel=2 m/s CPDAT239 Tool[4]:Microflown3D Base[2]:straight_sol;%{PE}
;FOLD Parameters ;%{h}
;Params IlfProvider=kukaroboter.basistech.inlineforms.movement.spline; Kuka.IsGlobalPoint=False; Kuka.PointName=P239; Kuka.BlendingEnabled=False; Kuka.MoveDataName=CPDAT239; Kuka.VelocityPath=2.000; Kuka.VelocityFieldEnabled=True; Kuka.ColDetectFieldEnabled=True; Kuka.CurrentCDSetIndex=0; Kuka.MovementParameterFieldEnabled=True; IlfCommand=SLIN
;ENDFOLD
SLIN XP239 WITH $VEL = SVEL_CP(2.0, , LCPDAT239),$TOOL = STOOL2(FP239),$BASE = SBASE(FP239.BASE_NO),$IPO_MODE = SIPO_MODE(FP239.IPO_FRAME),$LOAD = SLOAD(FP239.TOOL_NO),$ACC = SACC_CP(LCPDAT239),$ORI_TYPE = SORI_TYP(LCPDAT239),$APO = SAPO(LCPDAT239),$JERK = SJERK(LCPDAT239),$COLLMON_TOL_PRO[1] = USE_CM_PRO_VALUES(0)
;ENDFOLD

;FOLD SLIN P240 Vel=2 m/s CPDAT240 Tool[4]:Microflown3D Base[2]:straight_sol;%{PE}
;FOLD Parameters ;%{h}
;Params IlfProvider=kukaroboter.basistech.inlineforms.movement.spline; Kuka.IsGlobalPoint=False; Kuka.PointName=P240; Kuka.BlendingEnabled=False; Kuka.MoveDataName=CPDAT240; Kuka.VelocityPath=2.000; Kuka.VelocityFieldEnabled=True; Kuka.ColDetectFieldEnabled=True; Kuka.CurrentCDSetIndex=0; Kuka.MovementParameterFieldEnabled=True; IlfCommand=SLIN
;ENDFOLD
SLIN XP240 WITH $VEL = SVEL_CP(2.0, , LCPDAT240),$TOOL = STOOL2(FP240),$BASE = SBASE(FP240.BASE_NO),$IPO_MODE = SIPO_MODE(FP240.IPO_FRAME),$LOAD = SLOAD(FP240.TOOL_NO),$ACC = SACC_CP(LCPDAT240),$ORI_TYPE = SORI_TYP(LCPDAT240),$APO = SAPO(LCPDAT240),$JERK = SJERK(LCPDAT240),$COLLMON_TOL_PRO[1] = USE_CM_PRO_VALUES(0)
;ENDFOLD

;FOLD SLIN P241 Vel=2 m/s CPDAT241 Tool[4]:Microflown3D Base[2]:straight_sol;%{PE}
;FOLD Parameters ;%{h}
;Params IlfProvider=kukaroboter.basistech.inlineforms.movement.spline; Kuka.IsGlobalPoint=False; Kuka.PointName=P241; Kuka.BlendingEnabled=False; Kuka.MoveDataName=CPDAT241; Kuka.VelocityPath=2.000; Kuka.VelocityFieldEnabled=True; Kuka.ColDetectFieldEnabled=True; Kuka.CurrentCDSetIndex=0; Kuka.MovementParameterFieldEnabled=True; IlfCommand=SLIN
;ENDFOLD
SLIN XP241 WITH $VEL = SVEL_CP(2.0, , LCPDAT241),$TOOL = STOOL2(FP241),$BASE = SBASE(FP241.BASE_NO),$IPO_MODE = SIPO_MODE(FP241.IPO_FRAME),$LOAD = SLOAD(FP241.TOOL_NO),$ACC = SACC_CP(LCPDAT241),$ORI_TYPE = SORI_TYP(LCPDAT241),$APO = SAPO(LCPDAT241),$JERK = SJERK(LCPDAT241),$COLLMON_TOL_PRO[1] = USE_CM_PRO_VALUES(0)
;ENDFOLD

;FOLD SLIN P242 Vel=2 m/s CPDAT242 Tool[4]:Microflown3D Base[2]:straight_sol;%{PE}
;FOLD Parameters ;%{h}
;Params IlfProvider=kukaroboter.basistech.inlineforms.movement.spline; Kuka.IsGlobalPoint=False; Kuka.PointName=P242; Kuka.BlendingEnabled=False; Kuka.MoveDataName=CPDAT242; Kuka.VelocityPath=2.000; Kuka.VelocityFieldEnabled=True; Kuka.ColDetectFieldEnabled=True; Kuka.CurrentCDSetIndex=0; Kuka.MovementParameterFieldEnabled=True; IlfCommand=SLIN
;ENDFOLD
SLIN XP242 WITH $VEL = SVEL_CP(2.0, , LCPDAT242),$TOOL = STOOL2(FP242),$BASE = SBASE(FP242.BASE_NO),$IPO_MODE = SIPO_MODE(FP242.IPO_FRAME),$LOAD = SLOAD(FP242.TOOL_NO),$ACC = SACC_CP(LCPDAT242),$ORI_TYPE = SORI_TYP(LCPDAT242),$APO = SAPO(LCPDAT242),$JERK = SJERK(LCPDAT242),$COLLMON_TOL_PRO[1] = USE_CM_PRO_VALUES(0)
;ENDFOLD

;FOLD SLIN P243 Vel=2 m/s CPDAT243 Tool[4]:Microflown3D Base[2]:straight_sol;%{PE}
;FOLD Parameters ;%{h}
;Params IlfProvider=kukaroboter.basistech.inlineforms.movement.spline; Kuka.IsGlobalPoint=False; Kuka.PointName=P243; Kuka.BlendingEnabled=False; Kuka.MoveDataName=CPDAT243; Kuka.VelocityPath=2.000; Kuka.VelocityFieldEnabled=True; Kuka.ColDetectFieldEnabled=True; Kuka.CurrentCDSetIndex=0; Kuka.MovementParameterFieldEnabled=True; IlfCommand=SLIN
;ENDFOLD
SLIN XP243 WITH $VEL = SVEL_CP(2.0, , LCPDAT243),$TOOL = STOOL2(FP243),$BASE = SBASE(FP243.BASE_NO),$IPO_MODE = SIPO_MODE(FP243.IPO_FRAME),$LOAD = SLOAD(FP243.TOOL_NO),$ACC = SACC_CP(LCPDAT243),$ORI_TYPE = SORI_TYP(LCPDAT243),$APO = SAPO(LCPDAT243),$JERK = SJERK(LCPDAT243),$COLLMON_TOL_PRO[1] = USE_CM_PRO_VALUES(0)
;ENDFOLD

;FOLD SLIN P244 Vel=2 m/s CPDAT244 Tool[4]:Microflown3D Base[2]:straight_sol;%{PE}
;FOLD Parameters ;%{h}
;Params IlfProvider=kukaroboter.basistech.inlineforms.movement.spline; Kuka.IsGlobalPoint=False; Kuka.PointName=P244; Kuka.BlendingEnabled=False; Kuka.MoveDataName=CPDAT244; Kuka.VelocityPath=2.000; Kuka.VelocityFieldEnabled=True; Kuka.ColDetectFieldEnabled=True; Kuka.CurrentCDSetIndex=0; Kuka.MovementParameterFieldEnabled=True; IlfCommand=SLIN
;ENDFOLD
SLIN XP244 WITH $VEL = SVEL_CP(2.0, , LCPDAT244),$TOOL = STOOL2(FP244),$BASE = SBASE(FP244.BASE_NO),$IPO_MODE = SIPO_MODE(FP244.IPO_FRAME),$LOAD = SLOAD(FP244.TOOL_NO),$ACC = SACC_CP(LCPDAT244),$ORI_TYPE = SORI_TYP(LCPDAT244),$APO = SAPO(LCPDAT244),$JERK = SJERK(LCPDAT244),$COLLMON_TOL_PRO[1] = USE_CM_PRO_VALUES(0)
;ENDFOLD

;FOLD SLIN P245 Vel=2 m/s CPDAT245 Tool[4]:Microflown3D Base[2]:straight_sol;%{PE}
;FOLD Parameters ;%{h}
;Params IlfProvider=kukaroboter.basistech.inlineforms.movement.spline; Kuka.IsGlobalPoint=False; Kuka.PointName=P245; Kuka.BlendingEnabled=False; Kuka.MoveDataName=CPDAT245; Kuka.VelocityPath=2.000; Kuka.VelocityFieldEnabled=True; Kuka.ColDetectFieldEnabled=True; Kuka.CurrentCDSetIndex=0; Kuka.MovementParameterFieldEnabled=True; IlfCommand=SLIN
;ENDFOLD
SLIN XP245 WITH $VEL = SVEL_CP(2.0, , LCPDAT245),$TOOL = STOOL2(FP245),$BASE = SBASE(FP245.BASE_NO),$IPO_MODE = SIPO_MODE(FP245.IPO_FRAME),$LOAD = SLOAD(FP245.TOOL_NO),$ACC = SACC_CP(LCPDAT245),$ORI_TYPE = SORI_TYP(LCPDAT245),$APO = SAPO(LCPDAT245),$JERK = SJERK(LCPDAT245),$COLLMON_TOL_PRO[1] = USE_CM_PRO_VALUES(0)
;ENDFOLD

;FOLD SLIN P246 Vel=2 m/s CPDAT246 Tool[4]:Microflown3D Base[2]:straight_sol;%{PE}
;FOLD Parameters ;%{h}
;Params IlfProvider=kukaroboter.basistech.inlineforms.movement.spline; Kuka.IsGlobalPoint=False; Kuka.PointName=P246; Kuka.BlendingEnabled=False; Kuka.MoveDataName=CPDAT246; Kuka.VelocityPath=2.000; Kuka.VelocityFieldEnabled=True; Kuka.ColDetectFieldEnabled=True; Kuka.CurrentCDSetIndex=0; Kuka.MovementParameterFieldEnabled=True; IlfCommand=SLIN
;ENDFOLD
SLIN XP246 WITH $VEL = SVEL_CP(2.0, , LCPDAT246),$TOOL = STOOL2(FP246),$BASE = SBASE(FP246.BASE_NO),$IPO_MODE = SIPO_MODE(FP246.IPO_FRAME),$LOAD = SLOAD(FP246.TOOL_NO),$ACC = SACC_CP(LCPDAT246),$ORI_TYPE = SORI_TYP(LCPDAT246),$APO = SAPO(LCPDAT246),$JERK = SJERK(LCPDAT246),$COLLMON_TOL_PRO[1] = USE_CM_PRO_VALUES(0)
;ENDFOLD

;FOLD SLIN P247 Vel=2 m/s CPDAT247 Tool[4]:Microflown3D Base[2]:straight_sol;%{PE}
;FOLD Parameters ;%{h}
;Params IlfProvider=kukaroboter.basistech.inlineforms.movement.spline; Kuka.IsGlobalPoint=False; Kuka.PointName=P247; Kuka.BlendingEnabled=False; Kuka.MoveDataName=CPDAT247; Kuka.VelocityPath=2.000; Kuka.VelocityFieldEnabled=True; Kuka.ColDetectFieldEnabled=True; Kuka.CurrentCDSetIndex=0; Kuka.MovementParameterFieldEnabled=True; IlfCommand=SLIN
;ENDFOLD
SLIN XP247 WITH $VEL = SVEL_CP(2.0, , LCPDAT247),$TOOL = STOOL2(FP247),$BASE = SBASE(FP247.BASE_NO),$IPO_MODE = SIPO_MODE(FP247.IPO_FRAME),$LOAD = SLOAD(FP247.TOOL_NO),$ACC = SACC_CP(LCPDAT247),$ORI_TYPE = SORI_TYP(LCPDAT247),$APO = SAPO(LCPDAT247),$JERK = SJERK(LCPDAT247),$COLLMON_TOL_PRO[1] = USE_CM_PRO_VALUES(0)
;ENDFOLD

;FOLD SLIN P248 Vel=2 m/s CPDAT248 Tool[4]:Microflown3D Base[2]:straight_sol;%{PE}
;FOLD Parameters ;%{h}
;Params IlfProvider=kukaroboter.basistech.inlineforms.movement.spline; Kuka.IsGlobalPoint=False; Kuka.PointName=P248; Kuka.BlendingEnabled=False; Kuka.MoveDataName=CPDAT248; Kuka.VelocityPath=2.000; Kuka.VelocityFieldEnabled=True; Kuka.ColDetectFieldEnabled=True; Kuka.CurrentCDSetIndex=0; Kuka.MovementParameterFieldEnabled=True; IlfCommand=SLIN
;ENDFOLD
SLIN XP248 WITH $VEL = SVEL_CP(2.0, , LCPDAT248),$TOOL = STOOL2(FP248),$BASE = SBASE(FP248.BASE_NO),$IPO_MODE = SIPO_MODE(FP248.IPO_FRAME),$LOAD = SLOAD(FP248.TOOL_NO),$ACC = SACC_CP(LCPDAT248),$ORI_TYPE = SORI_TYP(LCPDAT248),$APO = SAPO(LCPDAT248),$JERK = SJERK(LCPDAT248),$COLLMON_TOL_PRO[1] = USE_CM_PRO_VALUES(0)
;ENDFOLD

;FOLD SLIN P249 Vel=2 m/s CPDAT249 Tool[4]:Microflown3D Base[2]:straight_sol;%{PE}
;FOLD Parameters ;%{h}
;Params IlfProvider=kukaroboter.basistech.inlineforms.movement.spline; Kuka.IsGlobalPoint=False; Kuka.PointName=P249; Kuka.BlendingEnabled=False; Kuka.MoveDataName=CPDAT249; Kuka.VelocityPath=2.000; Kuka.VelocityFieldEnabled=True; Kuka.ColDetectFieldEnabled=True; Kuka.CurrentCDSetIndex=0; Kuka.MovementParameterFieldEnabled=True; IlfCommand=SLIN
;ENDFOLD
SLIN XP249 WITH $VEL = SVEL_CP(2.0, , LCPDAT249),$TOOL = STOOL2(FP249),$BASE = SBASE(FP249.BASE_NO),$IPO_MODE = SIPO_MODE(FP249.IPO_FRAME),$LOAD = SLOAD(FP249.TOOL_NO),$ACC = SACC_CP(LCPDAT249),$ORI_TYPE = SORI_TYP(LCPDAT249),$APO = SAPO(LCPDAT249),$JERK = SJERK(LCPDAT249),$COLLMON_TOL_PRO[1] = USE_CM_PRO_VALUES(0)
;ENDFOLD

;FOLD SLIN P250 Vel=2 m/s CPDAT250 Tool[4]:Microflown3D Base[2]:straight_sol;%{PE}
;FOLD Parameters ;%{h}
;Params IlfProvider=kukaroboter.basistech.inlineforms.movement.spline; Kuka.IsGlobalPoint=False; Kuka.PointName=P250; Kuka.BlendingEnabled=False; Kuka.MoveDataName=CPDAT250; Kuka.VelocityPath=2.000; Kuka.VelocityFieldEnabled=True; Kuka.ColDetectFieldEnabled=True; Kuka.CurrentCDSetIndex=0; Kuka.MovementParameterFieldEnabled=True; IlfCommand=SLIN
;ENDFOLD
SLIN XP250 WITH $VEL = SVEL_CP(2.0, , LCPDAT250),$TOOL = STOOL2(FP250),$BASE = SBASE(FP250.BASE_NO),$IPO_MODE = SIPO_MODE(FP250.IPO_FRAME),$LOAD = SLOAD(FP250.TOOL_NO),$ACC = SACC_CP(LCPDAT250),$ORI_TYPE = SORI_TYP(LCPDAT250),$APO = SAPO(LCPDAT250),$JERK = SJERK(LCPDAT250),$COLLMON_TOL_PRO[1] = USE_CM_PRO_VALUES(0)
;ENDFOLD

;FOLD SLIN P251 Vel=2 m/s CPDAT251 Tool[4]:Microflown3D Base[2]:straight_sol;%{PE}
;FOLD Parameters ;%{h}
;Params IlfProvider=kukaroboter.basistech.inlineforms.movement.spline; Kuka.IsGlobalPoint=False; Kuka.PointName=P251; Kuka.BlendingEnabled=False; Kuka.MoveDataName=CPDAT251; Kuka.VelocityPath=2.000; Kuka.VelocityFieldEnabled=True; Kuka.ColDetectFieldEnabled=True; Kuka.CurrentCDSetIndex=0; Kuka.MovementParameterFieldEnabled=True; IlfCommand=SLIN
;ENDFOLD
SLIN XP251 WITH $VEL = SVEL_CP(2.0, , LCPDAT251),$TOOL = STOOL2(FP251),$BASE = SBASE(FP251.BASE_NO),$IPO_MODE = SIPO_MODE(FP251.IPO_FRAME),$LOAD = SLOAD(FP251.TOOL_NO),$ACC = SACC_CP(LCPDAT251),$ORI_TYPE = SORI_TYP(LCPDAT251),$APO = SAPO(LCPDAT251),$JERK = SJERK(LCPDAT251),$COLLMON_TOL_PRO[1] = USE_CM_PRO_VALUES(0)
;ENDFOLD

;FOLD SLIN P252 Vel=2 m/s CPDAT252 Tool[4]:Microflown3D Base[2]:straight_sol;%{PE}
;FOLD Parameters ;%{h}
;Params IlfProvider=kukaroboter.basistech.inlineforms.movement.spline; Kuka.IsGlobalPoint=False; Kuka.PointName=P252; Kuka.BlendingEnabled=False; Kuka.MoveDataName=CPDAT252; Kuka.VelocityPath=2.000; Kuka.VelocityFieldEnabled=True; Kuka.ColDetectFieldEnabled=True; Kuka.CurrentCDSetIndex=0; Kuka.MovementParameterFieldEnabled=True; IlfCommand=SLIN
;ENDFOLD
SLIN XP252 WITH $VEL = SVEL_CP(2.0, , LCPDAT252),$TOOL = STOOL2(FP252),$BASE = SBASE(FP252.BASE_NO),$IPO_MODE = SIPO_MODE(FP252.IPO_FRAME),$LOAD = SLOAD(FP252.TOOL_NO),$ACC = SACC_CP(LCPDAT252),$ORI_TYPE = SORI_TYP(LCPDAT252),$APO = SAPO(LCPDAT252),$JERK = SJERK(LCPDAT252),$COLLMON_TOL_PRO[1] = USE_CM_PRO_VALUES(0)
;ENDFOLD

